(* CoDeSys 2.3 project: cy-02-wg-030.pro *)
(* Title: cy-02-wg - Albino Infanzia E10 *)
(* Author: Andrea Ravasio *)
(* Libraries: Standard.lib 2.12.10 14:48:34, Util.lib 26.9.14 10:12:46, Visual.lib 2.12.10 14:48:34, WagoLibIdent.lib 25.2.13 11:12:16, WagoLibStatus.lib 2.12.10 14:48:32, SysLibFile.lib 2.12.10 14:48:34, SysLibRtc.lib 2.12.10 14:48:32, SysLibSockets.lib 10.2.11 09:20:54, SysLibEvent.lib 2.12.10 14:48:34, SysLibPlcCtrl.lib 2.12.10 14:48:32, SysLibCallback.lib 2.12.10 14:48:32, serial_interface_01.lib 22.4.13 12:50:14, SerComm.lib 31.5.11 08:54:36, MBus_03.lib 9.2.13 17:51:58, mod_com.lib 2.12.10 14:48:32, Modb_l05.lib 22.4.13 12:50:12 *)

(* PLC configuration (modules and I/O channels)
0750-1506 8DI / 8DO 24V DC 0.5A [Type_34_8_Channels] node 0, in %IB12 out %QB8 {INTTypePAAssignment = PLC; INTTypeModule = plugged}
  CIR06_AL AT %IX6.0 [BOOLOnX_I] Ch_1 Digital input
  CIR06_EN AT %QX4.0 [BOOLOnX_Q] 9 - Ch_1 Digital output
  CIR06_ST AT %IX6.1 [BOOLOnX_I] Ch_2 Digital input
  CIR06_ECO AT %QX4.1 [BOOLOnX_Q] 10 - Ch_2 Digital output
  CIR05_AL AT %IX6.2 [BOOLOnX_I] Ch_3 Digital input
  CIR05_EN AT %QX4.2 [BOOLOnX_Q] 11 - Ch_3 Digital output
  CIR06_AUTO AT %IX6.3 [BOOLOnX_I] Ch_4 Digital input
  CIR05_ECO AT %QX4.3 [BOOLOnX_Q] 12 - Ch_4 Digital output
  CIR04_AL AT %IX6.4 [BOOLOnX_I] Ch_5 Digital input
  CIR04_EN AT %QX4.4 [BOOLOnX_Q] 13 - Ch_5 Digital output
  CIR05_ST AT %IX6.5 [BOOLOnX_I] Ch_6 Digital input
  CIR04_ECO AT %QX4.5 [BOOLOnX_Q] 14 - Ch_6 Digital output
  CIR03_AL AT %IX6.6 [BOOLOnX_I] Ch_7 Digital input
  CIR03_EN AT %QX4.6 [BOOLOnX_Q] 15 - Ch_7 Digital output
  CIR05_AUTO AT %IX6.7 [BOOLOnX_I] Ch_8 Digital input
  CIR03_ECO AT %QX4.7 [BOOLOnX_Q] 16 - Ch_8 Digital output
0750-1506 8DI / 8DO 24V DC 0.5A [Type_34_8_Channels] node 1, in %IB12 out %QB8 {INTTypePAAssignment = PLC; INTTypeModule = plugged}
  CTL01_ST AT %IX6.8 [BOOLOnX_I] Ch_1 Digital input
  DOOR2_EN AT %QX4.8 [BOOLOnX_Q] 9 - Ch_1 Digital output
  DOOR2_ST AT %IX6.9 [BOOLOnX_I] Ch_2 Digital input
  CIR01_EN AT %QX4.9 [BOOLOnX_Q] 10 - Ch_2 Digital output
  CIR01_AL AT %IX6.10 [BOOLOnX_I] Ch_3 Digital input
  CIR02_EN AT %QX4.10 [BOOLOnX_Q] 11 - Ch_3 Digital output
  CIR01_ST AT %IX6.11 [BOOLOnX_I] Ch_4 Digital input
  AT %QX4.11 [BOOLOnX_Q] 12 - Ch_4 Digital output
  CIR03_ST AT %IX6.12 [BOOLOnX_I] Ch_5 Digital input
  AT %QX4.12 [BOOLOnX_Q] 13 - Ch_5 Digital output
  CIR01_AUTO AT %IX6.13 [BOOLOnX_I] Ch_6 Digital input
  AT %QX4.13 [BOOLOnX_Q] 14 - Ch_6 Digital output
  CIR02_AL AT %IX6.14 [BOOLOnX_I] Ch_7 Digital input
  AT %QX4.14 [BOOLOnX_Q] 15 - Ch_7 Digital output
  CIR02_ST AT %IX6.15 [BOOLOnX_I] Ch_8 Digital input
  AT %QX4.15 [BOOLOnX_Q] 16 - Ch_8 Digital output
0750-1506 8DI / 8DO 24V DC 0.5A [Type_34_8_Channels] node 2, in %IB13 out %QB9 {INTTypePAAssignment = PLC; INTTypeModule = plugged}
  KEY_CT_ST AT %IX7.0 [BOOLOnX_I] Ch_1 Digital input
  KEY_CT_EN AT %QX5.0 [BOOLOnX_Q] 9 - Ch_1 Digital output
  GZB_ST AT %IX7.1 [BOOLOnX_I] Ch_2 Digital input
  GZB_CTRL AT %QX5.1 [BOOLOnX_Q] 10 - Ch_2 Digital output
  VPN_OUT2 AT %IX7.2 [BOOLOnX_I] Ch_3 Digital input
  VPN_DIS AT %QX5.2 [BOOLOnX_Q] 11 - Ch_3 Digital output
  CIR04_AUTO AT %IX7.3 [BOOLOnX_I] Ch_4 Digital input
  AT %QX5.3 [BOOLOnX_Q] 12 - Ch_4 Digital output
  KEY_QE_ST AT %IX7.4 [BOOLOnX_I] Ch_5 Digital input
  AT %QX5.4 [BOOLOnX_Q] 13 - Ch_5 Digital output
  CIR03_AUTO AT %IX7.5 [BOOLOnX_I] Ch_6 Digital input
  AT %QX5.5 [BOOLOnX_Q] 14 - Ch_6 Digital output
  CIR02_AUTO AT %IX7.6 [BOOLOnX_I] Ch_7 Digital input
  TEST1 AT %QX5.6 [BOOLOnX_Q] 15 - Ch_7 Digital output
  CIR04_ST AT %IX7.7 [BOOLOnX_I] Ch_8 Digital input
  TEST2 AT %QX5.7 [BOOLOnX_Q] 16 - Ch_8 Digital output
0750-0650/0003-0000#03 RS 232 C Interface (Adjustable), 3 Byte [Type_21_1_Channels] node 3, in %IB8 out %QB8 {INTTypePAAssignment = PLC; INTTypeModule = plugged}
  AT %IX0.0 [BOOLOnX_I] Transmission acknowledgement
  AT %IX0.1 [BOOLOnX_I] Reception request
  AT %IX0.2 [BOOLOnX_I] Initialization acknowledgement
  AT %IX0.3 [BOOLOnX_I] Input buffer is full
  AT %IX0.4 [BOOLOnX_I] Number of received characters Bit 0
  AT %IX0.5 [BOOLOnX_I] Number of received characters Bit 1
  AT %IX0.6 [BOOLOnX_I] Number of received characters Bit 2
  AT %IB1 [BYTEOnB_I] Input data Byte 0
  AT %IB2 [BYTEOnB_I] Input data Byte 1
  AT %IB3 [BYTEOnB_I] Input data Byte 2
  AT %QX0.0 [BOOLOnX_Q] Transmission request
  AT %QX0.1 [BOOLOnX_Q] Reception acknowledgement
  AT %QX0.2 [BOOLOnX_Q] Initialization request
  AT %QX0.4 [BOOLOnX_Q] Number of characters Bit 0
  AT %QX0.5 [BOOLOnX_Q] Number of characters Bit 1
  AT %QX0.6 [BOOLOnX_Q] Number of characters Bit 2
  AT %QB1 [BYTEOnB_Q] Output data Byte 0
  AT %QB2 [BYTEOnB_Q] Output data Byte 1
  AT %QB3 [BYTEOnB_Q] Output data Byte 2
0750-0650/0003-0000#03 RS 232 C Interface (Adjustable), 3 Byte [Type_21_1_Channels] node 4, in %IB8 out %QB8 {INTTypePAAssignment = PLC; INTTypeModule = plugged}
  AT %IX2.0 [BOOLOnX_I] Transmission acknowledgement
  AT %IX2.1 [BOOLOnX_I] Reception request
  AT %IX2.2 [BOOLOnX_I] Initialization acknowledgement
  AT %IX2.3 [BOOLOnX_I] Input buffer is full
  AT %IX2.4 [BOOLOnX_I] Number of received characters Bit 0
  AT %IX2.5 [BOOLOnX_I] Number of received characters Bit 1
  AT %IX2.6 [BOOLOnX_I] Number of received characters Bit 2
  AT %IB5 [BYTEOnB_I] Input data Byte 0
  AT %IB6 [BYTEOnB_I] Input data Byte 1
  AT %IB7 [BYTEOnB_I] Input data Byte 2
  AT %QX2.0 [BOOLOnX_Q] Transmission request
  AT %QX2.1 [BOOLOnX_Q] Reception acknowledgement
  AT %QX2.2 [BOOLOnX_Q] Initialization request
  AT %QX2.4 [BOOLOnX_Q] Number of characters Bit 0
  AT %QX2.5 [BOOLOnX_Q] Number of characters Bit 1
  AT %QX2.6 [BOOLOnX_Q] Number of characters Bit 2
  AT %QB5 [BYTEOnB_Q] Output data Byte 0
  AT %QB6 [BYTEOnB_Q] Output data Byte 1
  AT %QB7 [BYTEOnB_Q] Output data Byte 2
0750-0461 2 AI PT100 (RTD) [Type_44_2_Channels] node 5, in %IB12 out %QB12 {INTTypePAAssignment = PLC; INTTypeModule = plugged}
  T_S02 AT %IW4 [INTOnW_I] Ch_1 signed Input value
  T_S01 AT %IW5 [INTOnW_I] Ch_2 signed Input value
Fieldbus variables [FB_VARS] node 1, in %IB0 out %QB0
Flag variables [FLAG_VARS] node 2, in %IB0 out %QB0
Modbus-Master [MB_MASTER] node 3, in %IB0 out %QB0
*)

(* Global variable list: Global_Constants *)
VAR_GLOBAL CONSTANT

	Plant_NAME			: STRING :='cySN:2 cyVER:30 - Albino Infanzia E10';
	Plant_SN			: DWORD  :=2;  		(* S/N Impianto di telecontrollo *)
	Plant_SW_VER		: WORD   :=30;		(* Versione SW installata *)

	(* Parameters *)
	Plant_DefaultTAmb	: INT	:=100;		(* [.1°C] Temperatura ambiente di default in caso di rottura sonda *)
	Plant_MaxRunTAmb	: INT   :=250; 		(* [.1°C] Temperatura ambiente massima funzionamento impianto *)
	Plant_AntiFreezeTAmb: INT   :=-40;		(* [.1°C] Antifreeze temperature, start circulators *)
	Plant_VRD_TAlarm	: INT   :=450; 		(* [.1°C] Temperatura di allarme VRD, blocco *)
	Plant_VRD_TMax		: INT   :=430; 		(* [.1°C] Setpoint massimo per uscita VRD *)
	Plant_VRD_TDefault	: INT	:=300;		(* [.1°C] Temperatura di default in caso di errore climatica *)
	Plant_CirOffDelay	: TIME	:=T#15m;	(* (Def.T#15m) Ritardo spegnimento pompe per ricircolo caldaia *)
	Plant_MaxWaterLoss	: WORD  :=2;		(* [lt/h] Massima perdita del circuito *)

	(* Filesystem *)
	FilesPath  			: STRING :='S:\';

	(* TCP Logger *)
	Logger_SERVER		: STRING:='';
	Logger_IP			: STRING:='192.168.100.3';
	Logger_PORT			: WORD  :=80;
	Logger_GETSTART		: STRING:='GET /cygmsrv/hsgm.ashx?';
	Logger_GETEND		: STRING:='$R$N$R$N';
	Logger_CHECK		: STRING:='True';
	Logger_CRLF			: STRING:='$R$N';
	Logger_DataFile		: STRING:='S:\LOG.DAT';
	Logger_DataFileOld	: STRING:='S:\LOG.BCK';
	Logger_IndexFile	: STRING:='S:\LOG.IDX';
	Logger_ConnRetries	: BYTE:=5;
	Logger_RecoverMsgs	: BYTE:=100;

	(* TCP Remote *)
	Remote_PORT			: WORD  :=10;
	Remote_WELCOME		: STRING:='Connected$R$N';
	Remote_OK			: STRING:='OK$R$N';
	Remote_ERROR		: STRING:='ERROR$R$N';

	(* TCP Sockets *)
	MAX_SEND_TCP_SERVER					 : DWORD:=3000;(*60000*)
	MAX_RECEIVE_TCP_SERVER				 : DWORD:=3000;
	MAX_RECEIVE_TCP_SERVER_SOCKET	 	 : DWORD:=1500;
	MAX_SEND_TCP_CLIENT					 : DWORD:=3000;(*15000*)
	MAX_RECEIVE_TCP_CLIENT				 : DWORD:=1500;
	MAX_RECEIVE_TCP_CLIENT_SOCKET		 : DWORD:=1500;
	MAX_RECEIVE_UDP_SERVER				 : INT  :=1472;
	MAX_RECEIVE_UDP_CLIENT				 : INT  :=1472;
	CONNECT_WATCHDOG_TIME				 : TIME :=t#10s;

	(* VISU COLORS *)
	COLOR_RED 		: DWORD:=16#2020F0;
	COLOR_YELLOW	: DWORD:=16#20F0F0;
	COLOR_GREEN		: DWORD:=16#20F020;
	COLOR_GREEN_OFF : DWORD:=16#006000;
	COLOR_LBLUE		: DWORD:=16#F0F080;

END_VAR

(* Global variable list: Global_Retain *)
VAR_GLOBAL RETAIN PERSISTENT
	GRU01_Clima : typ_Clima;
	CTL01_Count : DWORD;

	Mode_Manual : BOOL := FALSE;
END_VAR

(* Global variable list: Global_Variables *)
VAR_GLOBAL

	SYS    : typ_SYS;

	MODB01 : obj_MODBUS				:= ( ID:=1 , COM:=3, BAUDRATE:=BAUD_19200 );
	GRU01  : obj_MODBUS_ROBUR_DDC	:= ( ID:=1 , NetID:=479 );
	PDC01  : obj_PDC_ROBUR_GAHP		:= ( ID:=1 , NetID:=0 );
	CAL01  : obj_CAL_ROBUR_AY		:= ( ID:=1 , NetID:=1 );
	CAL02  : obj_CAL_ROBUR_AY		:= ( ID:=2 , NetID:=2 );

	TPV01  : obj_TPV				:= ( ID:=1 ); (* T_S01 - T_Amb *)
	TPV02  : obj_TPV				:= ( ID:=2 , IN_WMIN:=50 , IN_WMAX:=800 ); (* T_S02 *)
	TPV03  : obj_TPV				:= ( ID:=3 , IN_WMIN:=50 , IN_WMAX:=800 ); (* GRU01 - T_Send *)
	TPV04  : obj_TPV				:= ( ID:=4 , IN_WMIN:=50 , IN_WMAX:=800 ); (* GRU01 - T_Return *)
	TPV05  : obj_TPV				:= ( ID:=5 ); (* GRU01 - T_Amb *)
	T_AMB  : INT; (* From TPV01 *)

	CIR01  : obj_CIR				:= ( ID:=1 );
	CIR02  : obj_CIR				:= ( ID:=2 );
	CIR03  : obj_CIR				:= ( ID:=3 );
	CIR04  : obj_CIR				:= ( ID:=4 );
	CIR05  : obj_CIR				:= ( ID:=5 );
	CIR06  : obj_CIR				:= ( ID:=6 );

	CRON01 : obj_CRON				:= ( ID:=1 );
	CRON02 : obj_CRON				:= ( ID:=2 );
	CRON03 : obj_CRON				:= ( ID:=3 );
	CRON04 : obj_CRON				:= ( ID:=4 );
	CRON05 : obj_CRON				:= ( ID:=5 );
	CRON06 : obj_CRON				:= ( ID:=6 );
	CronEd : obj_CRON_EDITOR;

	CTL01  : obj_CTL				:= ( ID:=1 );

	MBUS01 : obj_MBUS				:= ( ID:=1 , COM:=2 , BAUDRATE:=BAUD_2400 );
	CTB01  : obj_MBUS_CTB			:= ( ID:=1 , ADDRESS:=0 );

	Logger : typ_Logger;

	(**** SIMULATION ONLY ****)
(*	CIR01_EN	:BOOL;
	CIR01_ST	:BOOL;
	CIR01_MAN	:BOOL;
	CIR01_AL	:BOOL:=TRUE;
	CIR03_EN	:BOOL;
	CIR03_ECO	:BOOL;
	CIR03_ST	:BOOL;
	CIR03_AL	:BOOL;
	CIR04_EN	:BOOL;
	CIR04_ECO	:BOOL;
	CIR04_ST	:BOOL;
	CIR04_AL	:BOOL;
	CIR05_EN	:BOOL;
	CIR05_ECO	:BOOL;
	CIR05_ST	:BOOL;
	CIR05_AL	:BOOL;
	CIR06_EN	:BOOL;
	CIR06_ECO	:BOOL;
	CIR06_ST	:BOOL;
	CIR06_AL	:BOOL;
	CTL01_ST	:BOOL;
	KEY_CT_ST	:BOOL;
	KEY_CT_EN	:BOOL;
	GZB_ST		:BOOL;
	GZB_CTRL	:BOOL;
	VPN_DIS		:BOOL;
	VPN_ST1		:BOOL:=TRUE;
	VPN_ST2		:BOOL;
	VPN_CTRL1	:BOOL;
	VPN_CTRL2	:BOOL;
	KEY_QE_ST	:BOOL:=TRUE;
(*	TEST1		:BOOL;	*)
	TEST2		:BOOL;
	T_S01		:INT:=100;
	T_S02		:INT:=100;
*)

END_VAR

(* Data type in Logger *)
TYPE en_Logger_ErrLev :
(
	EL_Log			:=0,
	EL_Wrn			:=1,
	EL_Alarm		:=2,
	EL_AlarmStop	:=3
);
END_TYPE

(* Data type in Logger *)
TYPE en_Logger_Status :
(
	S_Logger_UNKNOWN := 0,
	S_Logger_IDLE,
	S_Logger_WAITCONN,
	S_Logger_WAITTX,
	S_Logger_WAITRESP,
	S_Logger_ERROR
);
END_TYPE

(* Data type *)
TYPE en_SYS_Objects :
(
	EO_SYS		:=0,  (* PLC *)
	EO_VPN		:=1,  (* VPN *)
	EO_DOOR		:=2,  (* Door & access control *)

	EO_CAL		:=10, (* Caldaia *)
	EO_CIR		:=11, (* Circolatore *)
	EO_CRON		:=12, (* Crono-termostato *)
	EO_VRD		:=13, (* Valvola miscelatore pannelli *)
	EO_CTL		:=14, (* Contalitri *)
	EO_CTB		:=15, (* Contabilizzatore *)
	EO_TPV		:=16, (* Temperature probes values *)
	EO_PPV		:=17, (* Pressure probes values *)
	EO_PBV		:=18, (* Over-Pressure Alarms *)
	EO_TBV		:=19, (* Over-Temperature Alarms *)
	EO_PMV		:=20, (* Under-Pressure Alarms *)
	EO_GRU		:=21, (* Gruppo termico *)
	EO_PDC		:=22, (* Pompa di calore *)
	EO_SOL		:=23, (* Pannello solare termico *)
	EO_ESOL		:=24, (* Pannello solare fotovoltaico *)
	EO_GAS		:=25, (* Contatore GAS *)
	EO_PORT		:=26, (* Misuratore di portata *)
	EO_FPV		:=27, (* Flow probes values *)
	EO_ANZ		:=28, (* Analizzatore di rete *)
	EO_SCA		:=29, (* Signal Control Alarms *)
	EO_LUX		:=30, (* Base Illumination point *)
	EO_LUXM		:=31, (* Metered Illumination point *)
	EO_PSG		:=32, (* Sensore di passaggio *)
	EO_HVAC		:=33, (* Heating, Ventilating and Air Conditioning *)
	EO_HYGRV	:=34, (* Relative Humidity sensors value *)
	EO_COOV		:=35, (* Carbon Dioxide CO2 sensors value *)

	EO_ZGW			:=200,  (* ZigBee - Gateway *)
	EO_ZRM			:=201,	(* ZigBee - Repeater *)
	EO_ZREL			:=202,	(* ZigBee - Actuator rele *)
	EO_ZTHL			:=203,	(* ZigBee - Temperature Sensor *)

	EO_ASGW			:=250,	(* ASi - Gateway *)
	EO_ASCBI		:=251,	(* ASi - Input Board, Ciabatta *)

	EO_LON			:=1000, (* Bus - LON *)
	EO_MODBUS		:=1001, (* Bus - MODBUS *)
	EO_MBUS			:=1002, (* Bus - M-BUS *)
	EO_MODBUS_TCP	:=1003, (* Bus - MODBUS TCP *)

	EO_GENERIC		:=9000, (* Generic dataset *)
	EO_EXPO			:=9001  (* EXPO dataset *)
);
END_TYPE

(* Data type *)
TYPE en_SYS_Status :
(
	S_UNKNOWN  := 0,
	S_STARTUP,
	S_INIT_RTC,
	S_INIT_VAR,
	S_AUTOTEST,
	S_RUNNING,
	S_SHUTDOWN,
	S_HALT
);
END_TYPE

(* Data type in Plant_Objects *)
TYPE typ_Clima : (* CURVA CLIMATICA *)
STRUCT
	InitOK:		BOOL;
	Points: 	ARRAY [0..10] OF POINT;
END_STRUCT
END_TYPE

(* Data type in Plant_Objects *)
TYPE typ_Cron_Calendar :
STRUCT
	Profile		: ARRAY[0..384] OF BYTE;
END_STRUCT
END_TYPE

(* Data type in Plant_Objects *)
TYPE typ_Cron_Jolly :
STRUCT
	Start		: DT;
	End			: DT;
	Temp		: WORD;
	Flags		: WORD; (* B0:Enabled B1..B15:Unused *)
END_STRUCT
END_TYPE

(* Data type in Plant_Objects *)
TYPE typ_Cron_Profile :
STRUCT
	Flags		: WORD;
	Setpoint	: ARRAY [0..95] OF WORD;
END_STRUCT
END_TYPE

(* Data type in Logger *)
TYPE typ_Logger :
STRUCT
	Status		: en_Logger_Status;

	SendReq		: BOOL;
	SendIdx		: DWORD;
	SendData	: ARRAY [0..MAX_SEND_TCP_CLIENT] OF BYTE;
	SendLen		: DINT;

	TData		: ARRAY [0..MAX_SEND_TCP_CLIENT] OF BYTE;
	TLen		: DINT;

	LastIdxPos	: DWORD;

	(* Temporary variables used by objects *)
	s1			: STRING(256);
	i1			: WORD;

END_STRUCT
END_TYPE

(* Data type in Plant_Objects *)
TYPE typ_MODBUS_VAR : (* Gestione parametri MODBUS *)
STRUCT
	SlaveAddress	: BYTE;
	FunCode			: BYTE;
	FunAddress		: WORD;
	Refresh_Time	: BYTE; (* 0:No refresh x:Refresh in seconds *)
	Refresh_Cnt		: BYTE; (* INTERNAL *)
	Variable		: POINTER TO WORD;
	Variable_Size	: BYTE;
	Variable_Mirror : WORD; (* INTERNAL [Force refresh on read variables when <>0] *)
END_STRUCT
END_TYPE

(* Data type *)
TYPE typ_SYS :
STRUCT
	Status			: en_SYS_Status;
	Warning			: BOOL;
	Alarm			: BOOL;
	AlarmStop		: BOOL;

	Time_LogString	: STRING;
	Time_Year		: WORD;
	Time_Month		: BYTE;
	Time_Day		: BYTE;

	Time_CT_DT		: DT;
	Time_CT_Day		: WORD;
	Time_CT_Quarter	: BYTE;

	LastLogs_Idx	: BYTE;
	LastLogs_Dat	: ARRAY[0..5] OF STRING;
	LastLogs_Msg	: ARRAY[0..5] OF STRING;

END_STRUCT
END_TYPE

(* POU PLC_PRG, ST *)
PROGRAM PLC_PRG
VAR
	Timer1: TON; (* Fast controls tick *)
	Timer2: TON; (* Plant control tick *)
	Timer3: TON; (* Logger timer *)
END_VAR
(******************************************************************************
 ****                           MAIN TASK CODE                             ****
 ******************************************************************************

	Network setup:
		IP  = 192.168.100.2 | MSK = 255.255.255.0
		GW	= 192.168.100.1 | DNS = 192.168.100.1
		SNTP = 193.204.114.232 (3600s) ==> 192.168.100.3

*)

(*==============================*)
(*===== Main status machine ====*)
(*==============================*)
Main_Stm();

(*==============================*)
(*== Running cycle operations ==*)
(*==============================*)
IF SYS.Status>S_INIT_VAR THEN

	(* Execute MODBUS process *)
	MODB01();
	(* Execute M-BUS processes *)
	MBUS01();
	CTB01( MBus:=MBUS01.MBus );
	(*
	MBUS02();
	CTB02( MBus:=MBUS02.MBus );
	*)

END_IF

(*==============================*)
(*== System cycle operations ===*)
(*==============================*)
(* Execute TCP processes *)
Logger_Proc();
Remote_Proc();
(* Update user led *)
USRLED_Update();
(* Execute Cron Editor commands *)
CronEd();
(* External resources *)
   IF NOT TPV01.ERR THEN T_AMB:=T_S01;
ELSIF NOT TPV05.ERR THEN T_AMB:=GRU01.TAmb;
ELSE 					 T_AMB:=Plant_DefaultTAmb;
END_IF

(**** SIMULATION ONLY ****)
(*
CIR01_ST:=CIR01_EN XOR TEST2;
CIR03_ST:=CIR03_EN XOR TEST2;
CIR04_ST:=CIR04_EN XOR TEST2;
CIR05_ST:=CIR05_EN XOR TEST2;
CIR06_ST:=CIR06_EN XOR TEST2;
*)
END_PROGRAM
ACTION Main_Stm:
CASE Sys.Status OF

	S_STARTUP:
		Sys.Status:=S_INIT_RTC;

	S_INIT_RTC:
		(* Check RTC and update from network *)
		RTC_Update();
		(* Check time *)
		IF Sys.Time_Year>2000 THEN
			Sys.Status:=S_INIT_VAR;
		END_IF

	S_INIT_VAR:
		LogEv(EL_Wrn,EO_SYS,0,1,CONCAT('System_startup_v',WORD_TO_STRING(Plant_SW_VER)));
		Sys.Status:=S_RUNNING;

	S_RUNNING:
		Timer1(IN:=NOT Timer1.Q,PT:=T#50ms);
		IF Timer1.Q THEN
			(* Update meters *)
			CTL01 ( CTL_ST:=CTL01_ST, COUNT:=CTL01_Count );
			(* Update system checks *)
			SYS_Proc();
		END_IF

		Timer2(IN:=NOT Timer2.Q,PT:=T#500ms);
		IF Timer2.Q THEN
			(* Read current date/time *)
			RTC_Update();
			(* Execute plant operations *)
			TPV01	 ( IN:=T_S01 );
			TPV02	 ( IN:=T_S02 );
			TPV03	 ( IN:=GRU01.TSend );
			TPV04	 ( IN:=GRU01.TRet );
			TPV05	 ( IN:=GRU01.TAmb );
			(* CRON01   ( SETPOINT=>CIR01.Ctrl_SetPoint ); *) CRON01(); CIR01.CIR_RUN_REQ:=SEL(CRON01.SetPoint>180,FALSE,TRUE);
			(* CRON02   ( SETPOINT=>CIR02.Ctrl_SetPoint ); *) CRON02(); CIR02.CIR_RUN_REQ:=SEL(CRON02.SetPoint>180,FALSE,TRUE);
			CRON03   ( SETPOINT=>CIR03.Ctrl_SetPoint );
			CRON04   ( SETPOINT=>CIR04.Ctrl_SetPoint );
			CRON05   ( SETPOINT=>CIR05.Ctrl_SetPoint );
			CRON06   ( SETPOINT=>CIR06.Ctrl_SetPoint );
			CIR01    ( CIR_AL:=CIR01_AL , CIR_ST:=CIR01_ST , CIR_AUTO:=CIR01_AUTO , CIR_EN=>CIR01_EN );
			CIR02    ( CIR_AL:=CIR02_AL , CIR_ST:=CIR02_ST , CIR_AUTO:=CIR02_AUTO , CIR_EN=>CIR02_EN );
			CIR03    ( CIR_AL:=CIR03_AL , CIR_ST:=CIR03_ST , CIR_AUTO:=CIR03_AUTO , CIR_EN=>CIR03_EN );
			CIR04    ( CIR_AL:=CIR04_AL , CIR_ST:=CIR04_ST , CIR_AUTO:=CIR04_AUTO , CIR_EN=>CIR04_EN );
			CIR05    ( CIR_AL:=CIR05_AL , CIR_ST:=CIR05_ST , CIR_AUTO:=CIR05_AUTO , CIR_EN=>CIR05_EN );
			CIR06    ( CIR_AL:=CIR06_AL , CIR_ST:=CIR06_ST , CIR_AUTO:=CIR06_AUTO , CIR_EN=>CIR06_EN );
			GRU01.Run:=( CIR01.Run OR CIR03.Run OR CIR04.Run OR CIR05.Run OR CIR06.Run ) AND SYS.AlarmStop=FALSE;
			GRU01	 ( Clima:=GRU01_Clima, MODBUS:=MODB01 );
			PDC01	 ();
			CAL01	 ();
			CAL02	 ();
			(* Test toggle *)
			IF TEST1 THEN TEST1:=FALSE; ELSE TEST1:=TRUE; END_IF
		END_IF

		Timer3(IN:=NOT Timer3.Q,PT:=T#5m);
		IF Timer3.Q THEN
			(* Trig logger *)
			LogTrig();
			(* Execute temporary CSV logger *)
			CSV_Log();
		END_IF

	S_SHUTDOWN:
		(* Stop caldaia *)
		(* Stop deviatori *)
		(* Aspetta 5 min prima di spegnere eventuali circolatori *)
		Sys.Status:=S_STARTUP;

	S_HALT:
		(* Aspetta uscita manuale *)
		Sys.Status:=S_STARTUP;

ELSE
	Sys.Status:=S_STARTUP;
END_CASE;
END_ACTION

(* POU TCP_Logger/Logger_Proc, ST *)
PROGRAM Logger_Proc
VAR
	c1:         	TCPCLIENT;

	Open:	    	BOOL;
	IpAddr:			DWORD;
	InetAddr:		DWORD;
	Connected:  	BOOL;
	Error:      	DINT;
	TxTrig:     	BOOL;
	RxData:			ARRAY [0..MAX_RECEIVE_TCP_CLIENT] OF BYTE;
	RxLen:			DINT;

	Retry:			BYTE;	(* Counter for connection retries *)
	Recovered:		BYTE;	(* Counter for recovered unsent messages *)

	i:				DINT;
	pos:			DWORD;
	hFile:			DWORD;

END_VAR
(*=== State machine ===*)
CASE Logger.Status OF

	S_Logger_UNKNOWN:
		(* Startup *)
		Logger.SendReq:=FALSE;
		Open:=FALSE;
		Logger.Status:=S_Logger_IDLE;

	S_Logger_IDLE:
		(* Wait request *)
		IF Logger.SendReq THEN
			(* Resolve server name or use static IP *)
			IF LEN(Logger_SERVER)=0 THEN
				InetAddr:=SysSockInetAddr(Logger_IP);
			ELSE
				IpAddr:=SysSockGetHostByName(ADR(Logger_SERVER));
				DWORDSWAP(pIn:=ADR(IpAddr), pOut:=ADR(InetAddr));
			END_IF
			TxTrig:=FALSE;
			RxLen:=0;
			(* Open connection *)
			Open:=TRUE;
			Logger.Status:=S_Logger_WAITCONN;
		END_IF

	S_Logger_WAITCONN:
		(* Wait connection *)
		IF Connected THEN
			(* Send data *)
			TxTrig:=TRUE;
			Logger.Status:=S_Logger_WAITTX;
		END_IF
		IF Error>0 THEN
			Open:=FALSE;
			Logger.Status:=S_Logger_ERROR;
		END_IF

	S_Logger_WAITTX:
		(* Wait transmission *)
		IF NOT TxTrig THEN
			Logger.Status:=S_Logger_WAITRESP;
		END_IF
		IF Error>0 THEN
			Open:=FALSE;
			Logger.Status:=S_Logger_ERROR;
		END_IF

	S_Logger_WAITRESP:
		(* Wait response *)
		IF Connected=FALSE (* OR TIMEOUT!! *) THEN
			Open:=FALSE;
			(* Check response *)
			IF RxLen>=4 AND CHKSTRING(pString:=ADR(RxData), pPattern:=ADR(Logger_CHECK)) THEN
				Logger.SendReq:=FALSE;
				Retry:=0;
				(* Check unsent messages to flush *)
				IF Recovered<Logger_RecoverMsgs THEN
					MsgChk();
					IF Logger.SendReq=TRUE THEN
						Recovered:=Recovered+1;
					ELSE
						Recovered:=0;
					END_IF
				ELSE
					Recovered:=0;
				END_IF
				Logger.Status:=S_Logger_IDLE;
			ELSE
				Logger.Status:=S_Logger_ERROR;
			END_IF
		END_IF

	S_Logger_ERROR:
		(* Connection error or send failure *)
		Retry:=Retry+1;
		IF Retry>Logger_ConnRetries THEN
			(* Save message as unsent *)
			MsgSave();
			Logger.SendReq:=FALSE;
			Retry:=0;
		END_IF
		Logger.Status:=S_Logger_IDLE;

ELSE
	Logger.Status:=S_Logger_UNKNOWN;
END_CASE


(*=== Execute client lib ===*)
c1(
	xOpenConnection			:= Open,
	dwInetAddr 				:= InetAddr,
	wPortNumber				:= Logger_PORT,
	ptSendData				:= ADR(Logger.SendData),
	diSendCount				:= Logger.SendLen,
	tConnectWatchdogTime	:= t#10s,
	xStartSend				:= TxTrig,
	aReceiveBuffer			:= RxData,
	diReceiveCount			:= RxLen,
	xConnected				=> Connected,
	diError					=> Error
);

(*=== Process Rx data ===*)
(*IF RxLen>0 THEN
	RxLen:=0;
END_IF*)
END_PROGRAM
ACTION MsgChk:
(* Open index file *)
hFile:=SysFileOpen(Logger_IndexFile,'r');
IF hFile=0 THEN
	RETURN;
END_IF
(* Search oldest message to recover *)
SysFileSetPos(hFile,Logger.LastIdxPos);
Logger.SendLen:=0;
REPEAT
	SysFileRead(hFile, ADR(Logger.SendIdx), SIZEOF(Logger.SendIdx));
	pos:=SysFileGetPos(hFile);
	SysFileRead(hFile, ADR(Logger.SendLen), SIZEOF(Logger.SendLen));
UNTIL
	SysFileEOF(hFile) OR Logger.SendLen<>0
END_REPEAT
SysFileClose(hFile);
(* Delete index file when all messages are recovered *)
IF Logger.SendLen=0 THEN
	Logger.LastIdxPos:=0;
	SysFileDelete(Logger_IndexFile);
	RETURN;
END_IF
(* Recover message data *)
hFile:=SysFileOpen(Logger_DataFile,'r');
IF hFile<>0 THEN
	SysFileSetPos(hFile,Logger.SendIdx);
	SysFileRead(hFile,ADR(Logger.SendData),Logger.SendLen);
	Logger.SendReq:=TRUE;
	SysFileClose(hFile);
END_IF
(* Clear index entry *)
hFile:=SysFileOpen(Logger_IndexFile,'a');
IF hFile<>0 THEN
	SysFileSetPos(hFile,pos);
	i:=0;
	SysFileWrite(hFile, ADR(i), 4);
	Logger.LastIdxPos:=SysFileGetPos(hFile);
	SysFileClose(hFile);
END_IF
END_ACTION
ACTION MsgSave:
(* Add log position in recovery indexes *)
hFile:=SysFileOpen(Logger_IndexFile,'a');
SysFileWrite(hFile, ADR(Logger.SendIdx), SIZEOF(Logger.SendIdx));
SysFileWrite(hFile, ADR(Logger.SendLen), SIZEOF(Logger.SendLen));
SysFileClose(hFile);
END_ACTION

(* POU Utils Functions/TCPCLIENT, ST *)
FUNCTION_BLOCK TCPCLIENT
(***********************************************************************************************************	*)
(* Version: 1.3b                        			          													*)
(* Date: 28.10.2014                   				          							            			*)
(***********************************************************************************************************	*)
(* WAGO Kontakttechnik GmbH Hansastr. 27 32423 Minden(Westf.)													*)
(* Tel. +0049 571/887-0 Fax. +0049 571/887-0																	*)
(* Author: VB																									*)
(***********************************************************************************************************	*)
(*Description:	A TCP client to read and write data with additional connection watchdog							*)
(*History:																										*)
(*Version 1.3b: 28.10.2014: Use DWORD address for IP (Andrea Ravasio)											*)
(*Version 1.3: 11.02.2011: Changes according to 750-880/881											 			*)
(*Version 1.2: 29.08.2007 Bugfix TCP Client																		*)
(*Version 1.1: 15.01.2007 Changes according to FW11																*)
(*Version 1.0: 09.03.2006 Release																				*)
(***********************************************************************************************************	*)
VAR CONSTANT
	STATE_CREATE     				 : BYTE:= 0;
	STATE_OPEN     					 : BYTE:= 1;
	STATE_IOCTL    					 : BYTE:= 2;
	STATE_CONNECT     				 : BYTE:= 10;
	STATE_TX       					 : BYTE:= 20;
	STATE_RX       					 : BYTE:= 30;
	STATE_CLOSE    					 : BYTE:= 40;
	STATE_ERROR_TRAP			     : BYTE:= 200;
END_VAR

VAR_INPUT
	xOpenConnection					: BOOL;
	dwInetAddr						: DWORD; (* <== Use SysSockInetAddr() value or
													swapped bytes order of SysSockGetHostByName() value *)
	wPortNumber						: WORD;
	ptSendData						: POINTER TO ARRAY[0..MAX_SEND_TCP_CLIENT] OF BYTE;
	diSendCount						: DINT;
	tConnectWatchdogTime		    : TIME := t#10s;
END_VAR
VAR_OUTPUT
	xConnected						: BOOL;
	diError 						: DINT := 0;
END_VAR
(* ErrorCodes -----------------------------------------
	16#8001 => No socket descriptor available 
	16#8002 => SysSockSend returns -1 
	16#8003 => Socket was "gracefully closed" 
	16#8004 => switching to none blocking mode fails
	16#8005 => SysSockClose() returns FALSE 
    16#8006 => SysSockConnect() fails
    16#8007 => SysSockSend() fails
	16#8008 => error state machine 
	16#8009 => timeout while waiting for data from server 
------------------------------------------------------------*)
VAR_IN_OUT
	xStartSend							: BOOL;
	aReceiveBuffer						: ARRAY [0..MAX_RECEIVE_TCP_CLIENT] OF BYTE;
	diReceiveCount						: DINT;
END_VAR
VAR
	m_State								: BYTE := 0;
	m_ReceiveBuffer						: ARRAY [0..MAX_RECEIVE_TCP_CLIENT_SOCKET] OF BYTE;
	m_Socket							: DINT;
	m_AddressInfo						: SOCKADDRESS;
	m_BytesReceived						: DINT;
	m_diReturn							: DINT;
	m_xReturn							: BOOL;
	m_IoCtlParameter  					: DINT := 1; (* IOCTL-Parameter for non-blocking mode of sockets *)
	i									: INT;
	T_Connect							: TON;
	m_count								: DINT;
	diOption							: DINT := 1;
	m_Blocking   						: DINT := 0;
END_VAR
IF xOpenConnection THEN
	(* State maschine *)
	CASE  m_State OF

	(* -------------------------------------------------------------------------*)
	STATE_CREATE:
			(* create socket descriptor*)
			m_Socket := SysSockCreate(diAddressFamily	:= SOCKET_AF_INET,
													 diType		:= SOCKET_STREAM,
													 diProtocol := SOCKET_IPPROTO_TCP);
			IF m_Socket >= 0 THEN
			(*Set Push-Bit*)
				IF ADR(%MW0)=16#30000000  OR ADR(%MW0)=16#20000000 THEN (*841 or 881*)
					SysSockSetOption(
						diSocket:=m_Socket,
						diLevel:=6,
						diOption:=SOCKET_TCP_NODELAY,
						pOptionValue:=ADR(diOption),
						diOptionLength:=SIZEOF(diOption));
				ELSE
						;
				END_IF
				m_State := STATE_IOCTL; (* succesful *)
			ELSE
				diError := 16#8001;  (* no socket descriptor available *)
				m_State := STATE_ERROR_TRAP;
			END_IF

	(* -------------------------------------------------------------------------*)
	STATE_IOCTL: (* change  socket mode  to none blocking *)
		m_diReturn := SysSockIoctl( m_Socket, SOCKET_FIONBIO, ADR(m_IoCtlParameter));
		IF m_diReturn <> 0 THEN
			m_AddressInfo.sin_family := SOCKET_AF_INET;
			m_AddressInfo.sin_port := SysSockNtohs(wPortNumber);
			m_AddressInfo.sin_addr := dwInetAddr;
			m_State := STATE_CONNECT;
		ELSE
			diError := 16#8004;  (* switching to none blocking mode fails *)
			m_State := STATE_ERROR_TRAP;
		END_IF


	(* -------------------------------------------------------------------------*)
	STATE_CONNECT: (* connect with server *)
		T_Connect(IN:=TRUE , PT:=tConnectWatchdogTime);(*activate watchdog for establishing connection to a server*)
		m_xReturn := SysSockConnect ( m_Socket, ADR(m_AddressInfo),  SIZEOF(m_AddressInfo));
		IF m_xReturn THEN (* succesful *)
			IF xStartSend THEN
				m_State := STATE_TX;(*transmit data*)
			ELSE
				m_State := STATE_RX;(*wait for data from server*)
			END_IF
			xConnected:=TRUE;
			T_Connect(IN:=FALSE);
		ELSE
			IF T_Connect.Q THEN
				diError := 16#8006;  (* connect fails *)
				xConnected:=FALSE;
				T_Connect(IN:=FALSE);
				m_State := STATE_ERROR_TRAP;
				SysSockClose( m_Socket);
			ELSE
				m_State := STATE_CONNECT;(*client still  tries to set up connection*)
			END_IF
		END_IF


	STATE_TX:	 (* send TCP-message *)
		m_diReturn := SysSockSend(diSocket := m_Socket,
								  pbyBuffer := ADR(ptSendData^[0]),
								  diBufferSize := diSendCount-m_count,
								  diFlags := 0);

		CASE m_diReturn OF
		-1:	(* ERROR *)
			T_Connect(IN:=TRUE , PT:=CONNECT_WATCHDOG_TIME);(*activate watchdog to check communication*)
			IF t_Connect.Q THEN
				diError := 16#8007;
				T_Connect(IN:=FALSE);
				m_State:=STATE_CLOSE;
			END_IF
		0: (* socket was "gracefully closed" *)
			m_State := STATE_CLOSE;
			diError := 16#8003;
		ELSE (* succesful *)
			m_count:=m_count+m_diReturn;
			IF m_count>=diSendCount THEN
				diError := 16#0000;
				m_State := STATE_RX;
				m_count:=0;
				xStartSend:=FALSE;
			END_IF
			T_Connect(IN:=FALSE);
		END_CASE

	(* -------------------------------------------------------------------------*)
	STATE_RX: (* process receive data *)
			m_BytesReceived := SysSockRecv(	diSocket 	:= m_Socket,
										pbyBuffer 	:= ADR(m_ReceiveBuffer),		(* Address of receive buffer *)
										diBufferSize:= SIZEOF(m_ReceiveBuffer),
										diFlags		:= 0);

			CASE m_BytesReceived OF
			-1:	(* No data available or error occured *)
				T_Connect(IN:=TRUE , PT:=tConnectWatchdogTime);(*activate watchdog to check communication*)
				IF t_Connect.Q THEN
					diError:=16#8009;
					T_Connect(IN:=FALSE);
					m_State:=STATE_CLOSE;
				END_IF
				IF xStartSend THEN
					m_State:=STATE_TX	;(* WAIT IN THIS STATE  and check for arriving data or new send command*)
				END_IF;
			0: (* socket was "gracefully closed"  *)
				m_State:=STATE_CLOSE;
				diError := 16#8003;
			ELSE (* succesful *)
				diError := 16#0000;
				T_Connect(IN:=FALSE);
				(* Copy received data into receive buffer *)
				FOR i:= 0 TO DINT_TO_INT(m_BytesReceived	)-1 DO
					aReceiveBuffer[diReceiveCount]:= m_ReceiveBuffer[i];
					diReceiveCount:=(diReceiveCount+1) MOD SIZEOF(aReceiveBuffer);
				END_FOR

			END_CASE

	(* -------------------------------------------------------------------------*)
	STATE_CLOSE : (* close socket *)
		IF ADR(%MW0)=16#30000000  OR ADR(%MW0)=16#20000000 THEN (*841 or 881*)
			;
		ELSE
			SysSockShutdown(m_Socket, 0);;(*870*)
		END_IF
		m_xReturn := SysSockClose( m_Socket);
		m_Socket := -1;
		m_State := 0; (* succesful *)
		xConnected:=FALSE;
		T_Connect(IN:=FALSE);
	(* -------------------------------------------------------------------------*)
	STATE_ERROR_TRAP: (* error handling *)
		xConnected:=FALSE;

	ELSE  (* Bad FSM code trap  *)
			m_State:= STATE_ERROR_TRAP;
			diError:= 16#8008;
	END_CASE

ELSE(*close connection*)
	IF m_Socket >= 0 THEN
		IF ADR(%MW0)=16#30000000  OR ADR(%MW0)=16#20000000 THEN (*841 or 881*)
			;
		ELSE
			SysSockShutdown(m_Socket, 0);;(*870*)
		END_IF
		SysSockClose( m_Socket);
	END_IF
	m_Socket := -1;
	diError := 16#0000;
	m_State := STATE_CREATE;
	xConnected:=FALSE;
	T_Connect(IN:=FALSE);
END_IF
END_FUNCTION_BLOCK

(* POU Utils Functions/DWORDSWAP, ST *)
FUNCTION DWORDSWAP:BOOL
VAR_INPUT
	pIn:POINTER TO ARRAY[1..4] OF BYTE;
	pOut:POINTER TO ARRAY[1..4] OF BYTE;
END_VAR
VAR
END_VAR
pOut^[1]:=pIn^[4];
pOut^[2]:=pIn^[3];
pOut^[3]:=pIn^[2];
pOut^[4]:=pIn^[1];
END_FUNCTION

(* POU Utils Functions/CHKSTRING, ST *)
FUNCTION CHKSTRING : BOOL
VAR_INPUT
	pString: POINTER TO BYTE;
	pPattern: POINTER TO BYTE;
END_VAR
VAR
END_VAR
CHKSTRING:=TRUE;
WHILE pPattern^<>0 AND CHKSTRING DO
	IF pPattern^<>pString^ THEN CHKSTRING:=FALSE; END_IF
	pString:=pString+1;
	pPattern:=pPattern+1;
END_WHILE
END_FUNCTION

(* POU TCP_Remote/Remote_Proc, ST *)
PROGRAM Remote_Proc
VAR
	s1:         	TCPSERVER;
	Enable: 		BOOL;
	Connected: 		BOOL;
	Error: 			DINT;

	TxData:			ARRAY [0..MAX_SEND_TCP_SERVER] OF BYTE;
	TxLen:			DINT;
	TxTrig:			BOOL;

	RxData:			ARRAY [0..MAX_RECEIVE_TCP_SERVER] OF BYTE;
	RxLen:			DINT;

	Status:			DINT;

	(* Command interpreter *)

	Cmd_Buf:		ARRAY [0..MAX_RECEIVE_TCP_SERVER] OF BYTE;
	Cmd_Buf_U16:	POINTER TO WORD;
	Cmd_Buf_INT:	POINTER TO INT;
	Cmd_BufLen:		WORD;
	Cmd_St:			WORD;

	Cmd_Obj:		WORD;
	Cmd_ObjIdx:		WORD;
	Cmd_C:			WORD;
	Cmd_R:			WORD;
	Cmd_CLen:		WORD;
	Cmd_RLen:		WORD;

	i : WORD;
	j : INT;
	(*s2 : STRING;*)

END_VAR
(*=== State machine ===*)
CASE Status OF
	0: (* Startup *)
		TxLen:=0; TxTrig:=FALSE;
		RxLen:=0;
		Enable:=TRUE;
		Status:=1;

	1: (* Wait incoming connection *)
		IF Connected THEN
			(* Log access *)(*
			LogEv(EL_Log,EO_VPN,1,5,'Remote');*)
			(* Send welcome message *)(*
			ADDSTRING(pTxData:=ADR(TxData), pString:=ADR(Remote_WELCOME), TxLen:=TxLen);
			TxTrig:=TRUE;*)
			(* Reset vars *)
			Cmd_BufLen:=0;
			Cmd_St:=0;
			Status:=2;
		END_IF
		IF Error>1 THEN
			Enable:=FALSE;
			Status:=0;
		END_IF

	2: (* Wait command *)
		IF RxLen>0 THEN
			(*=== Interpreter start ===*)
			IF Cmd_BufLen+(RxLen/2)>=MAX_RECEIVE_TCP_SERVER THEN
				(* ERROR *)
				Cmd_BufLen:=0;
			ELSE
				i:=HEXTORAW(pString:=ADR(RxData), StringLen:=DINT_TO_WORD(RxLen), pData:=ADR(Cmd_Buf[Cmd_BufLen]));
				Cmd_BufLen:=Cmd_BufLen+i;
			END_IF
			IF Cmd_BufLen>=8 THEN
				Cmd_Buf_U16:=ADR(Cmd_Buf[6]);
				IF Cmd_BufLen>=(8+Cmd_Buf_U16^) THEN
					Cmd_CLen:=Cmd_Buf_U16^;
					Cmd_Buf_U16:=ADR(Cmd_Buf[0]); Cmd_Obj:=Cmd_Buf_U16^;
					Cmd_Buf_U16:=ADR(Cmd_Buf[2]); Cmd_ObjIdx:=Cmd_Buf_U16^;
					Cmd_Buf_U16:=ADR(Cmd_Buf[4]); Cmd_C:=Cmd_Buf_U16^;
					(* Log command *)(*
					s2:='RCmd_';		s2:=CONCAT(s2,WORD_TO_STRING(Cmd_Obj));
					s2:=CONCAT(s2,'_'); s2:=CONCAT(s2,WORD_TO_STRING(Cmd_ObjIdx));
					s2:=CONCAT(s2,'_'); s2:=CONCAT(s2,WORD_TO_STRING(Cmd_C));
					s2:=CONCAT(s2,'_');	s2:=CONCAT(s2,WORD_TO_STRING(Cmd_CLen));
					LogEv(EL_Log,EO_VPN,1,6,s2);*)
					(* Execute command *)
					Command();
					Cmd_BufLen:=0;
				END_IF
			END_IF
			(*=== Interpreter end ===*)
			RxLen:=0;
		END_IF
		IF NOT Connected THEN
			Status:=0;
		END_IF

ELSE
	Status:=0;
END_CASE


(*=== Execute server lib ===*)
s1(
	xEnable				:= Enable,
	wPortNumber			:= Remote_PORT,
	tServerTimeOut		:= t#15m,
	ptSendData			:= ADR(TxData),
	diSendCount			:= TxLen,
	xStartSend			:= TxTrig,
	aReceiveBuffer		:= RxData,
	diReceiveCount		:= RxLen,
	xClientConnected	=> Connected,
	diError				=> Error
);
END_PROGRAM
ACTION Cmd_CAL:
(* Check index *)
IF Cmd_ObjIdx<1 OR Cmd_ObjIdx>2 THEN
	Cmd_R:=2;
	RETURN;
END_IF

(* Process command *)
CASE Cmd_C OF

	3: (* TRY REARM *)
		IF Cmd_ObjIdx=1 THEN
			CAL01.Rearm:=TRUE;
		ELSE
			CAL02.Rearm:=TRUE;
		END_IF

ELSE
	Cmd_R:=3;
END_CASE
END_ACTION
ACTION Cmd_CRON:
(* Check index *)
IF Cmd_ObjIdx<1 OR Cmd_ObjIdx>6 THEN
	Cmd_R:=2;
	RETURN;
END_IF

(* Process command *)
CASE Cmd_C OF

	1: (* GET PROFILE *)
		IF Cmd_CLen<>3 THEN
			Cmd_R:=4;
		ELSE
			(* Load profile *)
			CronEd.CN_Sel:=WORD_TO_BYTE(Cmd_ObjIdx);
			Cmd_Buf_U16:=ADR(Cmd_Buf[8]);
			CronEd.CN_YSel:=Cmd_Buf_U16^;
			CronEd.PR_Sel:=Cmd_Buf[10];
			CronEd.PR_Load_Exe();
			(* Copy data *)
			Cmd_RLen:=192;
			TxLen:=TxLen+RAWTOHEX(ADR(CronEd.PR.Setpoint),192,ADR(TxData[TxLen]));
		END_IF

	2: (* SET PROFILE *)
		IF Cmd_CLen<>(3+192) THEN
			Cmd_R:=4;
		ELSE
			(* Save profile *)
			CronEd.CN_Sel:=WORD_TO_BYTE(Cmd_ObjIdx);
			Cmd_Buf_U16:=ADR(Cmd_Buf[8]);
			CronEd.CN_YSel:=Cmd_Buf_U16^;
			CronEd.PR_Sel:=Cmd_Buf[10];
			MEMCPY(ADR(Cmd_Buf[11]),ADR(CronEd.PR.Setpoint),192);
			CronEd.PR_Save_Exe();
		END_IF

	5: (* GET CALENDAR MONTH *)
		IF Cmd_CLen<>3 THEN
			Cmd_R:=4;
		ELSE
			(* Load calendar *)
			CronEd.CN_Sel:=WORD_TO_BYTE(Cmd_ObjIdx);
			Cmd_Buf_U16:=ADR(Cmd_Buf[8]);
			CronEd.CN_YSel:=Cmd_Buf_U16^;
			CronEd.CA_Sel:=Cmd_Buf[10];
			CronEd.CA_Load_Exe();
			(* Copy data *)
			Cmd_RLen:=32;
			TxLen:=TxLen+RAWTOHEX(ADR(CronEd.CA.Profile),32,ADR(TxData[TxLen]));
		END_IF

	6: (* SET CALENDAR MONTH *)
		IF Cmd_CLen<>(3+32) THEN
			Cmd_R:=4;
		ELSE
			(* Save calendar *)
			CronEd.CN_Sel:=WORD_TO_BYTE(Cmd_ObjIdx);
			Cmd_Buf_U16:=ADR(Cmd_Buf[8]);
			CronEd.CN_YSel:=Cmd_Buf_U16^;
			CronEd.CA_Sel:=Cmd_Buf[10];
			MEMCPY(ADR(Cmd_Buf[11]),ADR(CronEd.CA.Profile),32);
			CronEd.CA_Save_Exe();
		END_IF

	9: (* CRON RESTART *)
		CASE Cmd_ObjIdx OF
			1: CRON01.InitOK:=FALSE;
			2: CRON02.InitOK:=FALSE;
			3: CRON03.InitOK:=FALSE;
			4: CRON04.InitOK:=FALSE;
			5: CRON05.InitOK:=FALSE;
			6: CRON06.InitOK:=FALSE;
		END_CASE

ELSE
	Cmd_R:=3;
END_CASE
END_ACTION
ACTION Cmd_GRU:
(* Check index *)
IF Cmd_ObjIdx<>1 THEN
	Cmd_R:=2;
	RETURN;
END_IF

(* Process command *)
CASE Cmd_C OF

	1: (* GET CLIMATIC *)
		Cmd_RLen:=20;
		FOR i:=0 TO 4 DO
			j:=DINT_TO_INT(GRU01_Clima.Points[i].X);
			TxLen:=TxLen+RAWTOHEX(ADR(j),2,ADR(TxData[TxLen]));
			j:=DINT_TO_INT(GRU01_Clima.Points[i].Y);
			TxLen:=TxLen+RAWTOHEX(ADR(j),2,ADR(TxData[TxLen]));
		END_FOR

	2: (* SET CLIMATIC *)
		IF Cmd_CLen<>20 THEN
			Cmd_R:=4;
		ELSE
			FOR i:=0 TO 4 DO
				Cmd_Buf_INT:=ADR(Cmd_Buf[8+4*i]); j:=Cmd_Buf_INT^;
				GRU01_Clima.Points[i].X:=INT_TO_DINT(j);
				Cmd_Buf_INT:=ADR(Cmd_Buf[10+4*i]); j:=Cmd_Buf_INT^;
				GRU01_Clima.Points[i].Y:=INT_TO_DINT(j);
			END_FOR
		END_IF

ELSE
	Cmd_R:=3;
END_CASE
END_ACTION
ACTION Cmd_PDC:
(* Check index *)
IF Cmd_ObjIdx<>1 THEN
	Cmd_R:=2;
	RETURN;
END_IF

(* Process command *)
CASE Cmd_C OF

	3: (* TRY REARM *)
		PDC01.Rearm:=TRUE;

ELSE
	Cmd_R:=3;
END_CASE
END_ACTION
ACTION Cmd_SYS:
(* Check index *)
IF Cmd_ObjIdx<>0 THEN
	Cmd_R:=2;
	RETURN;
END_IF

(* Process command *)
CASE Cmd_C OF

	0: (* ECHO *)
		IF Cmd_CLen<>0 THEN
			TxLen:=0;
		END_IF

	1: (* LOG REQUEST *)
		LogTrig();

	2: (* REARM *)
		Sys.Warning:=FALSE;
		Sys.Alarm:=FALSE;
		Sys.AlarmStop:=FALSE;

	3: (* GET INFO1 *)
		Cmd_RLen:=6;
		TxLen:=TxLen+RAWTOHEX(ADR(Plant_SN),4,ADR(TxData[TxLen]));
		TxLen:=TxLen+RAWTOHEX(ADR(Plant_SW_VER),2,ADR(TxData[TxLen]));

ELSE
	Cmd_R:=3;
END_CASE
END_ACTION
ACTION Command:
(* Default response OK/NODATA *)
Cmd_R:=0;
Cmd_RLen:=0;
TxLen:=16;

(* Check object *)
CASE Cmd_Obj OF

	EO_SYS:
		Cmd_SYS();

	EO_GRU:
		Cmd_GRU();

	EO_PDC:
		Cmd_PDC();

	EO_CAL:
		Cmd_CAL();

	EO_CRON:
		Cmd_CRON();

ELSE
	Cmd_R:=1;
END_CASE

(* Generate response *)
IF TxLen>0 THEN
	RAWTOHEX(ADR(Cmd_Obj)	,2,ADR(TxData[ 0]));
	RAWTOHEX(ADR(Cmd_ObjIdx),2,ADR(TxData[ 4]));
	RAWTOHEX(ADR(Cmd_R)		,2,ADR(TxData[ 8]));
	RAWTOHEX(ADR(Cmd_RLen)	,2,ADR(TxData[12]));
	TxTrig:=TRUE;
END_IF
END_ACTION

(* POU Utils Functions/TCPSERVER, ST *)
FUNCTION_BLOCK TCPSERVER
(***********************************************************************************************************	*)
(* Version: 1.6                                    			          											*)
(* Date: 11.02.2011                                   					          							    *)
(***********************************************************************************************************	*)
(* WAGO Kontakttechnik GmbH Hansastr. 27 32423 Minden(Westf.)													*)
(* Tel. +0049 571/887-0 Fax. +0049 571/887-0																	*)
(* Author: VB																									*)
(***********************************************************************************************************	*)
(*Description:	A TCP server to read and write data													       		*)
(*Historie:																										*)
(*Version 1.6: 11.02.2011: Changes according to 750-880/881											 			*)
(*Version 1.5: 27.11.2008 Bugfix allow reuse port																*)
(*Version 1.4: 13.10.2008 Bugfix transmitting large data														*)
(*Version 1.3: 15.01.2007 Changes according to FW11																*)
(*Version 1.2: 09.03.2006 Changes for socket handle 0											       			*)
(*Version 1.1: 14.02.2005 Release																				*)
(***********************************************************************************************************	*)
VAR CONSTANT
	STATE_INIT     				 : BYTE:= 0;
	STATE_OPEN     				 : BYTE:= 1;
	STATE_TX       				 : BYTE:= 20;
	STATE_RX       				 : BYTE:= 30;
	STATE_CLOSE    				 : BYTE:= 40;
	STATE_ERROR_TRAP		 	 : BYTE:= 200;
END_VAR
VAR_INPUT
	xEnable    					: BOOL;	 (* Set TRUE to enable function block *)
	wPortNumber					: WORD;  (* Port *)
	tServerTimeOut				: TIME:=t#50s;
	ptSendData					: POINTER TO ARRAY[0..MAX_SEND_TCP_SERVER] OF BYTE;
	diSendCount					: DINT;
END_VAR
VAR_OUTPUT
	xClientConnected  			: BOOL:= FALSE;
	diError 					: DINT:= 0;
END_VAR
(* Status Codes -----------------------------------------
	16#8001 => No socket descriptor available 
	16#8002 => SysSockBind fails 
	16#8003 => SysSockListen fails 
	16#8004 => switching to none blocking mode fails
	16#8005 => SysSockClose() returns FALSE 
    16#8006 => SysSockConnect() fails
    16#8007 => SysSockSend() fails
	16#8008 => error state machine 
	16#8009 => timeout while waiting for data from server 
	16#0001 => server waiting for client to establish connection
------------------------------------------------------------*)
VAR_IN_OUT
	xStartSend					: BOOL;
	aReceiveBuffer				: ARRAY [0..MAX_RECEIVE_TCP_SERVER] OF BYTE;
	diReceiveCount				: DINT;
END_VAR

VAR
	m_State    					: BYTE:= 0;
	m_ReceiveBuffer				: ARRAY [0..MAX_RECEIVE_TCP_SERVER_SOCKET] OF BYTE;
	m_ServerSocket				: DINT:= SOCKET_INVALID;
	m_Socket					: DINT:= SOCKET_INVALID;
	m_AddressInfo				: SOCKADDRESS;
	m_BytesReceived				: DINT;
	m_diReturn					: DINT;
	m_xReturn					: BOOL;
	m_SizeSockadr				: DWORD;
	m_ConnectionWatchdog		: TON;
	m_Flags						: DINT;
	m_NoneBlocking   			: DINT:= 1;
	m_Blocking   				: DINT:= 0;
	i							: INT;
	m_count						: DINT;
	diOption					: DINT := 1;
	on: DINT;
END_VAR
IF xEnable THEN
	CASE m_State OF
		STATE_INIT:
			(* Create Socket *)
			m_ServerSocket:= SysSockCreate( SOCKET_AF_INET, SOCKET_STREAM, 0);
			IF m_ServerSocket = SOCKET_INVALID THEN
				(* *)
				diError:= 16#8001;
				m_State:= STATE_ERROR_TRAP;
				RETURN;
			ELSE
				;
			END_IF
			(* Address bindings *)
			(********************)
			on:=1;
			SysSockSetOption( m_ServerSocket, SOCKET_SOL, SOCKET_SO_REUSEADDR, ADR(on), SIZEOF(on) );

			m_AddressInfo.sin_family:= SOCKET_AF_INET;
			m_AddressInfo.sin_port  := SysSockHtons( wPortNumber);
			m_AddressInfo.sin_addr  := SOCKET_INADDR_ANY;
			IF NOT SysSockBind( m_ServerSocket, ADR(m_AddressInfo), SIZEOF(m_AddressInfo)) THEN
				diError:= 16#8002;
				m_State:= STATE_ERROR_TRAP;
				RETURN;
			END_IF
			(* Wait for connections *)
			(************************)
			IF NOT SysSockListen( m_ServerSocket, 1) THEN
				diError:= 16#8003;
				m_State:= STATE_ERROR_TRAP;
			END_IF

			(* Puts SOCKET in NonBlocking mode *)
			m_diReturn:= SysSockIoctl( m_ServerSocket, SOCKET_FIONBIO, ADR(m_NoneBlocking));

			m_State:= STATE_OPEN;


		STATE_OPEN: 	(* Waiting for incomming connection *)
				m_SizeSockadr:=SIZEOF(m_AddressInfo);
				m_Socket:= SysSockAccept( m_ServerSocket, ADR(m_AddressInfo), ADR(m_SizeSockadr));
				diError:=State_open;
				IF m_Socket <> SOCKET_INVALID THEN
					xClientConnected:=TRUE;
					(*Set Push-Bit:new V1.5*)
					IF ADR(%MW0)=16#30000000  OR ADR(%MW0)=16#20000000 THEN (*841 or 881*)
						SysSockSetOption(
							diSocket:=m_Socket,
							diLevel:=6,
							diOption:=SOCKET_TCP_NODELAY,
							pOptionValue:=ADR(diOption),
							diOptionLength:=SIZEOF(diOption));
					ELSE
							;
					END_IF
					SysSockIoctl( m_Socket, SOCKET_FIONBIO, ADR(m_NoneBlocking));
					m_State:= STATE_RX;
					diError:=0;
				END_IF

		STATE_RX:
					m_BytesReceived:= SysSockRecv( m_Socket, ADR(m_ReceiveBuffer), SIZEOF(m_ReceiveBuffer), 0);
					CASE m_BytesReceived OF
					-1:(*no data available or error occured*)
						m_ConnectionWatchdog(IN:=TRUE , PT:=tServerTimeOut );
						IF m_connectionWatchdog.Q THEN
							m_State:= STATE_CLOSE;
							m_ConnectionWatchdog(IN:=FALSE);(*reset connection watchdog*)
							diError := 16#8009;
						END_IF
					0:(* socket was "gracefully closed"  *)
						m_State:= STATE_CLOSE;
						diError := 16#8003;
					ELSE
						(* Copy received data into receive buffer *)
						(********************************)
						FOR i:= 0 TO DINT_TO_INT(m_BytesReceived	)-1 DO
							aReceiveBuffer[diReceiveCount]:= m_ReceiveBuffer[i];
							diReceiveCount:=(diReceiveCount+1) MOD SIZEOF(aReceiveBuffer);
						END_FOR

						m_ConnectionWatchdog(IN:=FALSE);(*reset connection watchdog*)
					END_CASE

				(*send data*)
				IF xStartSend	 THEN
					m_State := STATE_TX;
				END_IF

	STATE_TX:	 (* send TCP-message *)
		m_diReturn := SysSockSend(diSocket := m_Socket,
								  pbyBuffer := ADR(ptSendData^[m_count]),(*geändert V1.4 bisher: [0] *)
								  diBufferSize := diSendCount-m_count,
								  diFlags :=m_Flags);
		CASE m_diReturn OF
		-1:	(* ERROR or data could not yet be send (V1.3 due to new FW11) *)
			m_ConnectionWatchdog(IN:=TRUE , PT:=tServerTimeOut );
			IF m_connectionWatchdog.Q THEN
				m_State:= STATE_CLOSE;
				m_ConnectionWatchdog(IN:=FALSE);(*reset connection watchdog*)
				diError := 16#8007;
			END_IF
		0: (* socket was "gracefully closed"  *)
			m_State := STATE_CLOSE;
			diError := 16#8003;
		ELSE (* succesful *)
			m_count:=m_count+m_diReturn;
			IF m_count>=diSendCount THEN
				diError := 16#0000;
				m_State := STATE_RX;
				m_count:=0;
				xStartSend:=FALSE;
			END_IF
			m_ConnectionWatchdog(IN:=FALSE);(*reset connection watchdog*)
		END_CASE


		STATE_CLOSE:	(* Close the server *)

		IF ADR(%MW0)=16#30000000  OR ADR(%MW0)=16#20000000 THEN (*841 or 881*)
			;
		ELSE
			IF m_Socket>=0 THEN
				SysSockShutdown(m_Socket, 0);;(*870*)
			END_IF
		END_IF
		IF m_Socket>=0 THEN
			SysSockClose( m_Socket);
		END_IF
		xClientConnected:= FALSE;
		m_State:= STATE_OPEN; (* Try to open the server again *)
		m_ConnectionWatchdog(IN:=FALSE);(*reset connection watchdog*)

		STATE_ERROR_TRAP: (* Error Read/Write socket  *)
			m_State:= STATE_ERROR_TRAP;

	ELSE  (* Bad FSM code trap  *)
			m_State:= STATE_ERROR_TRAP;
			diError:= 16#8008;
	END_CASE;
ELSE
	IF m_State <> STATE_INIT THEN
		IF ADR(%MW0)=16#30000000  OR ADR(%MW0)=16#20000000 THEN (*841 or 881*)
			;
		ELSE
			IF m_Socket>=0 THEN
				SysSockShutdown(m_Socket, 0);;(*870*)
			END_IF
		END_IF
		IF m_Socket>=0 THEN
			SysSockClose( m_Socket);
		END_IF
		IF ADR(%MW0)=16#30000000  OR ADR(%MW0)=16#20000000 THEN (*841 or 881*)
			;
		ELSE
			IF m_ServerSocket>=0 THEN
				SysSockShutdown(m_ServerSocket, 0);;(*870*)
			END_IF
		END_IF
		IF m_ServerSocket>=0 THEN
			SysSockClose( m_ServerSocket);
		END_IF
		xClientConnected:= FALSE;
		diError:= 0;
		m_State:= STATE_init; (* Try to open the server again *)
		m_ConnectionWatchdog(IN:=FALSE);(*reset connection watchdog*)
	END_IF
END_IF
END_FUNCTION_BLOCK

(* POU Utils Functions/HEXTORAW, ST *)
FUNCTION HEXTORAW : WORD
VAR_INPUT
	pString		: POINTER TO BYTE;
	StringLen	: WORD;
	pData		: POINTER TO BYTE;
END_VAR
VAR
	xl: WORD;
	xi: WORD;
	xr: BYTE;
END_VAR
xl:=0;
xi:=0;

WHILE xi<StringLen DO

	IF pString^>=97 AND pString^<=102 THEN
		xr := pString^ - 87;
	ELSIF pString^>=65 AND pString^<=70 THEN
		xr := pString^ - 55;
	ELSIF pString^>=48 AND pString^<=57 THEN
		xr := pString^ - 48;
	ELSE
		xr := 16;
	END_IF

	IF xr<16 THEN
		IF (xi AND 1)=0 THEN
			pData^ := xr * 16;
		ELSE
			pData^ := pData^ + xr;
			pData := pData + 1;
			xl := xl + 1;
		END_IF
	END_IF

	xi := xi + 1;
	pString := pString + 1;

END_WHILE

HEXTORAW:=xl;
END_FUNCTION

(* POU Utils Functions/RAWTOHEX, ST *)
FUNCTION RAWTOHEX : WORD
VAR_INPUT
	pData: POINTER TO BYTE;
	DataLen: WORD;
	pString: POINTER TO BYTE;
END_VAR
VAR
	xl: WORD;
END_VAR
xl:=0;

WHILE DataLen>0 DO

	pString^ := (pData^ / 16#10) + 48 + (((pData^ / 16#10)/10)*7);
	pString:=pString+1;
	pString^ := (pData^ AND 16#0F)  + 48 + (((pData^ AND 16#0F)/10)*7);
	pString:=pString+1;
	pData:=pData+1;
	DataLen:=DataLen-1;
	xl:=xl+2;

END_WHILE

(*pString^:=0;*)

RAWTOHEX:=xl;
END_FUNCTION

(* POU Utils/USRLED_Update, ST *)
PROGRAM USRLED_Update
VAR
	OldStatus: en_SYS_Status;

	aFS : ARRAY [0..24] OF FLASHING_SEQUENCE :=
		(Colour:=GREEN,  Frequency:=1,   Relation:=128, Duration:=t#0s,    NextIndex:=0),  (* 0 => RUNNING *)
		(Colour:=ORANGE, Frequency:=1,   Relation:=128, Duration:=t#0s,    NextIndex:=1),  (* 1 => INIT *)
		(Colour:=RED,    Frequency:=4,   Relation:=128, Duration:=t#0s,    NextIndex:=2),  (* 2 => ERROR *)
		(Colour:=RED,    Frequency:=10,  Relation:=128, Duration:=t#0s,    NextIndex:=3),  (* 3 => ALARM *)
		(Colour:=ORANGE, Frequency:=200, Relation:=16,  Duration:=t#100ms, NextIndex:=11), (* 10 *)
		(Colour:=ORANGE, Frequency:=200, Relation:=32,  Duration:=t#100ms, NextIndex:=12),
		(Colour:=ORANGE, Frequency:=200, Relation:=64,  Duration:=t#100ms, NextIndex:=13),
		(Colour:=ORANGE, Frequency:=200, Relation:=128, Duration:=t#100ms, NextIndex:=14),
		(Colour:=ORANGE, Frequency:=200, Relation:=192, Duration:=t#100ms, NextIndex:=15),
		(Colour:=ORANGE, Frequency:=200, Relation:=128, Duration:=t#100ms, NextIndex:=16),
		(Colour:=ORANGE, Frequency:=200, Relation:=64,  Duration:=t#100ms, NextIndex:=17),
		(Colour:=ORANGE, Frequency:=200, Relation:=32,  Duration:=t#100ms, NextIndex:=18),
		(Colour:=ORANGE, Frequency:=200, Relation:=16,  Duration:=t#100ms, NextIndex:=19),
		(Colour:=ORANGE, Frequency:=200, Relation:=8,   Duration:=t#100ms, NextIndex:=10),
		(Colour:=GREEN,  Frequency:=200, Relation:=16,  Duration:=t#100ms, NextIndex:=21), (* 20 *)
		(Colour:=GREEN,  Frequency:=200, Relation:=32,  Duration:=t#100ms, NextIndex:=22),
		(Colour:=GREEN,  Frequency:=200, Relation:=64,  Duration:=t#100ms, NextIndex:=23),
		(Colour:=GREEN,  Frequency:=200, Relation:=128, Duration:=t#100ms, NextIndex:=24),
		(Colour:=GREEN,  Frequency:=200, Relation:=192, Duration:=t#100ms, NextIndex:=25),
		(Colour:=GREEN,  Frequency:=200, Relation:=128, Duration:=t#100ms, NextIndex:=26),
		(Colour:=GREEN,  Frequency:=200, Relation:=64,  Duration:=t#100ms, NextIndex:=27),
		(Colour:=GREEN,  Frequency:=200, Relation:=32,  Duration:=t#100ms, NextIndex:=28),
		(Colour:=GREEN,  Frequency:=200, Relation:=16,  Duration:=t#100ms, NextIndex:=29),
		(Colour:=GREEN,  Frequency:=200, Relation:=8,   Duration:=t#100ms, NextIndex:=20);

	pFS : POINTER TO FLASHING_SEQUENCE;


END_VAR
IF Sys.Status <> OldStatus THEN

	OldStatus:=Sys.Status;

	CASE OldStatus OF

		S_STARTUP:
			pFS:=ADR(aFS);
			SET_FLASHING_SEQUENCE(EN:=TRUE, POINTER_TO_POINTER_TO_ARRAY:=ADR(pFS));
			SET_FLASHING_SEQUENCE_INDEX(EN:=TRUE, IMMEDIATE:=FALSE, INDEX:=1);
			START_FLASHING_SEQUENCE(EN:=TRUE);

		S_RUNNING:
			SET_FLASHING_SEQUENCE_INDEX(EN:=TRUE, IMMEDIATE:=TRUE, INDEX:=0);

	END_CASE

END_IF
END_PROGRAM

(* POU Plant/SYS_Proc, ST *)
PROGRAM SYS_Proc
VAR
(*	fALARM_PB		:FLT_TAP;
	fALARM_TB		:FLT_TAP;
	fALARM_PM		:FLT_TAP; *)

(*	fGZB_ST			:FLT_TAP; (* GATEWAY ZIGBEE *)*)
(*	fVPN_OUT1		:FLT_TAP; (* VPN - CONNECT *)*)
	fVPN_OUT2		:FLT_TAP; (* VPN - STATUS *)
(*	fKEY_CT_ST		:FLT_TAP; (* DOOR01 - Porta primaria *)*)
(*	fKEY_SCT_ST		:FLT_TAP; (* DOOR02 - Porta secondaria *)*)
	fKEY_QE_ST		:FLT_TAP; (* DOOR03 - Quadro Elettrico *)

END_VAR
(*************** ISPESL *****************)
(*
fALARM_PB(IN:=ALARM_PB);
IF fALARM_PB.EVH THEN
	LogEv(EL_AlarmStop,EO_PBV,1,1,'Over_Pressure_Alarm');
END_IF

fALARM_TB(IN:=ALARM_TB);
IF fALARM_TB.EVH THEN
	LogEv(EL_AlarmStop,EO_TBV,1,1,'Over_Temperature_Alarm');
END_IF

fALARM_PM(IN:=ALARM_PM);
IF fALARM_PM.EVH THEN
	LogEv(EL_AlarmStop,EO_PMV,1,1,'Under_Pressure_Alarm');
END_IF
*)
(****************************************)

(*### VPN Connection Check ###*)(*
fVPN_OUT1(IN:=VPN_OUT1);
IF fVPN_OUT1.EVH THEN
	LogEv(EL_Log,EO_VPN,1,1,'CONNECT_ON');
END_IF
IF fVPN_OUT1.EVL THEN
	LogEv(EL_Log,EO_VPN,1,2,'CONNECT_OFF');
END_IF*)

(*### VPN Status Check ###*)
fVPN_OUT2(IN:=VPN_OUT2);
IF fVPN_OUT2.EVH THEN
	LogEv(EL_Log,EO_VPN,1,3,'STATUS_UP');
END_IF
IF fVPN_OUT2.EVL THEN
	LogEv(EL_Wrn,EO_VPN,1,4,'STATUS_DOWN');
END_IF

(*### DOOR01 Status Check ###*)(*
fKEY_CT_ST(IN:=KEY_CT_ST);
IF fKEY_CT_ST.EVH THEN
	LogEv(EL_Log,EO_DOOR,1,2,'Centrale_termica_Close');
END_IF
IF fKEY_CT_ST.EVL THEN
	LogEv(EL_Wrn,EO_DOOR,1,1,'Centrale_termica_Open');
END_IF*)

(*### DOOR02 Status Check ###*)(*
fKEY_SCT_ST(IN:=KEY_SCT_ST);
IF fKEY_SCT_ST.EVH THEN
	LogEv(EL_Log,EO_DOOR,2,2,'Sottocentrale_termica_Close');
END_IF
IF fKEY_SCT_ST.EVL THEN
	LogEv(EL_Wrn,EO_DOOR,2,1,'Sottocentrale_termica_Open');
END_IF*)

(*### DOOR03 Status Check ###*)
fKEY_QE_ST(IN:=KEY_QE_ST);
IF fKEY_QE_ST.EVH THEN
	LogEv(EL_Log,EO_DOOR,3,2,'Quadro_Close');
END_IF
IF fKEY_QE_ST.EVL THEN
	LogEv(EL_Wrn,EO_DOOR,3,1,'Quadro_Open');
END_IF
END_PROGRAM

(* POU Utils Functions/FLT_TAP, ST *)
FUNCTION_BLOCK FLT_TAP
VAR_INPUT
	IN		: BOOL;
	TAP		: BYTE:=4;
	INITEV	: BOOL:=TRUE;
END_VAR
VAR_OUTPUT
	OUT		: BOOL;
	EVH		: BOOL;
	EVL		: BOOL;
END_VAR
VAR
	init	: BOOL:=FALSE;
	cnt		: BYTE;
END_VAR
EVH:=FALSE;
EVL:=FALSE;

IF NOT init THEN
	init := TRUE;
	IF INITEV THEN
		OUT  := NOT IN;
		cnt  := TAP;
	ELSE
		OUT  := IN;
	END_IF
END_IF

IF OUT<>IN THEN
	cnt:=cnt+1;
	IF cnt>TAP THEN
		OUT:=IN;
		cnt:=0;
		IF OUT THEN EVH:=TRUE; ELSE EVL:=TRUE; END_IF
	END_IF
ELSE
	cnt:=0;
END_IF
END_FUNCTION_BLOCK

(* POU TCP_Logger/LogEv, ST *)
FUNCTION LogEv : BOOL
VAR_INPUT
	Level	: en_Logger_ErrLev;
	Object  : en_SYS_Objects;
	Index	: WORD;
	Error	: WORD;
	Message : STRING;
END_VAR
VAR
	s1 : STRING(160);
	i  : INT;
END_VAR
(* Execute error level operations *)
CASE Level OF
	EL_Wrn: 		Sys.Warning:=TRUE;
	EL_Alarm: 		Sys.Alarm  :=TRUE;
	EL_AlarmStop: 	Sys.Alarm  :=TRUE; (* GO TO STOP STATE!! *)
END_CASE

(* Fill lastlog list *)
s1:=CONCAT(Sys.Time_LogString,';Lev=');
s1:=CONCAT(s1,INT_TO_STRING(Level));
s1:=CONCAT(s1,';Obj=');
s1:=CONCAT(s1,INT_TO_STRING(Object));
s1:=CONCAT(s1,';Idx=');
s1:=CONCAT(s1,WORD_TO_STRING(Index));
s1:=CONCAT(s1,';Err=');
s1:=CONCAT(s1,WORD_TO_STRING(Error));
Sys.LastLogs_Dat[Sys.LastLogs_Idx]:=s1;
Sys.LastLogs_Msg[Sys.LastLogs_Idx]:=Message;
Sys.LastLogs_Idx:=Sys.LastLogs_Idx+1;
IF Sys.LastLogs_Idx>5 THEN Sys.LastLogs_Idx:=0; END_IF

(*---------------------------------------------------------------*)
	Logger_Head();
(*---------------------------------------------------------------*)

(* Insert ERR *)
s1:=CONCAT('&ERR=',INT_TO_STRING(Level));
s1:=CONCAT(s1,';');
s1:=CONCAT(s1,INT_TO_STRING(Object));
s1:=CONCAT(s1,';');
s1:=CONCAT(s1,WORD_TO_STRING(Index));
s1:=CONCAT(s1,';');
s1:=CONCAT(s1,WORD_TO_STRING(Error));
s1:=CONCAT(s1,';');
ADDSTRING(ADR(Logger.TData), ADR(s1), Logger.TLen);
s1:=Message;
STR_NOSPACES(ADR(s1));
ADDSTRING(ADR(Logger.TData), ADR(s1), Logger.TLen);

(*---------------------------------------------------------------*)
	Logger_Send();
(*---------------------------------------------------------------*)
END_FUNCTION

(* POU TCP_Logger/Logger_Head, ST *)
FUNCTION Logger_Head : BOOL
VAR
	s1 : STRING(160);
	i  : BYTE;
END_VAR
Logger.TLen:=0;
(* Set GET header *)
ADDSTRING(ADR(Logger.TData), ADR(Logger_GETSTART), Logger.TLen);

(* Insert Header *)
s1:=INSERT('ID=&V=1&D=',DWORD_TO_STRING(Plant_SN),3);
s1:=CONCAT(s1,Sys.Time_LogString);
s1:=CONCAT(s1,'&S=');
IF Sys.Alarm THEN i:=2; ELSIF Sys.Warning THEN i:=1; ELSE i:=0; END_IF
s1:=CONCAT(s1,BYTE_TO_STRING(i));
ADDSTRING(ADR(Logger.TData), ADR(s1), Logger.TLen);
END_FUNCTION

(* POU Utils Functions/ADDSTRING, ST *)
FUNCTION ADDSTRING : BOOL (* Append string to a byte buffer *)
VAR_INPUT
	pTxData: POINTER TO BYTE;
	pString: POINTER TO BYTE;
END_VAR
VAR_IN_OUT
	TxLen: DINT;
END_VAR
VAR
END_VAR
pTxData:=pTxData+TxLen;
WHILE pString^<>0 DO
	pTxData^:=pString^;
	pString:=pString+1;
	pTxData:=pTxData+1;
	TxLen:=TxLen+1;
END_WHILE
END_FUNCTION

(* POU Utils Functions/STR_NOSPACES, ST *)
FUNCTION STR_NOSPACES : BOOL (* Replace spaces and bad chars with allowed ones, used as HTTP-GET validator *)
VAR_INPUT
	pString: POINTER TO BYTE;
END_VAR
VAR
END_VAR
WHILE pString^<>0 DO
	IF pString^=16#20 (* space *) THEN pString^:=16#5F; (*'_'*) END_IF
	pString:=pString+1;
END_WHILE
END_FUNCTION

(* POU TCP_Logger/Logger_Send, ST *)
FUNCTION Logger_Send : BOOL
VAR
	hFile: 	DWORD;
	pos:	DWORD;
END_VAR
(* Finalize string *)
ADDSTRING(ADR(Logger.TData), ADR(Logger_GETEND), Logger.TLen);

(* Read log position *)
pos:=SysFileGetSize(Logger_DataFile);
(* Check log size, bckup and erase if no pending messages *)
IF pos>10000000 (*10M*) THEN
	hFile:=SysFileOpen(Logger_IndexFile,'r');
	IF hFile=0 THEN
		SysFileDelete(Logger_DataFileOld);
		SysFileRename(Logger_DataFile,Logger_DataFileOld);
		pos:=0;
	ELSE
		SysFileClose(hFile);
	END_IF
END_IF
(* Write message on log file *)
hFile:=SysFileOpen(Logger_DataFile,'a');
IF hFile<>0 THEN
	SysFileWrite(hFile, ADR(Logger.TData), Logger.TLen);
	SysFileClose(hFile);
ELSE
	Sys.Warning:=TRUE;
END_IF


(* Check logger status *)
IF Logger.SendReq=FALSE THEN
	(* Set log position for recovery *)
	Logger.SendIdx:=pos;
	(* Copy message data *)
	MEMCPY(ADR(Logger.TData),ADR(Logger.SendData),DINT_TO_WORD(Logger.TLen));
	Logger.SendLen:=Logger.TLen;
	(* Trigger request *)
	Logger.SendReq:=TRUE;
ELSE
	(* Add message position+size in recovery indexes *)
	hFile:=SysFileOpen(Logger_IndexFile,'a');
	SysFileWrite(hFile, ADR(pos), SIZEOF(pos));
	SysFileWrite(hFile, ADR(Logger.TLen), SIZEOF(Logger.TLen));
	SysFileClose(hFile);
END_IF
END_FUNCTION

(* POU Utils Functions/MEMCPY, ST *)
FUNCTION MEMCPY:BOOL
VAR_INPUT
	pSourceAddress:POINTER TO ARRAY[1..2] OF BYTE;
	pDestinationAddress:POINTER TO ARRAY[1..2] OF BYTE;
	BytesToCopy:WORD;
END_VAR
VAR
END_VAR
WHILE (BytesToCopy > 0) DO
	pDestinationAddress^[1]:=pSourceAddress^[1]; (* copy bytes from source to destination *)
	pDestinationAddress:=ADR(pDestinationAddress^[2]); (* increment destination *)
	pSourceAddress:=ADR(pSourceAddress^[2]);(* increment source *)
	BytesToCopy:=BytesToCopy -1; (* decrement number of bytes to copy *)
END_WHILE
END_FUNCTION

(* POU Utils Functions/AVERAGE_T, ST *)
FUNCTION_BLOCK AVERAGE_T
VAR_INPUT
	IN: 	INT;
END_VAR
VAR_OUTPUT
	HI:		INT;
	AVG:	INT;
	LOW:	INT;
	ERR:	BOOL;
END_VAR
VAR
	sum:	DINT;
	cnt:	WORD;
END_VAR
IF cnt>=65000 THEN
	ERR:=TRUE;
	Read();
	sum := sum - AVG;
	cnt := cnt + 1;
END_IF

sum := sum + IN;
cnt := cnt + 1;

IF IN<LOW THEN  LOW:=IN; END_IF
IF IN>HI  THEN HI :=IN; END_IF
END_FUNCTION_BLOCK
ACTION Read:
AVG := DINT_TO_INT(sum/cnt);
END_ACTION
ACTION Reset:
HI:=IN;
AVG:=IN;
LOW:=IN;
ERR:=FALSE;

sum:=IN;
cnt:=1;
END_ACTION

(* POU Utils Functions/COPY_32SWAP16, ST *)
FUNCTION COPY_32SWAP16:BOOL
VAR_INPUT
	pSourceAddress		:POINTER TO ARRAY[1..2] OF WORD;
	pDestinationAddress	:POINTER TO ARRAY[1..2] OF WORD;
END_VAR
VAR
END_VAR
pDestinationAddress^[1]:=pSourceAddress^[2];
pDestinationAddress^[2]:=pSourceAddress^[1];
END_FUNCTION

(* POU Utils/CSV_Log, ST *)
FUNCTION CSV_Log : BOOL
VAR_INPUT
END_VAR
VAR CONSTANT
	LogFileName:STRING:='S:\LOGS_ID2V3.CSV';
END_VAR
VAR
	s1 : STRING(256);
	hFile: 	DWORD;
END_VAR
(* Check file presence *)
hFile:=SysFileOpen(LogFileName,'r');
IF hFile=0 THEN
	(*** File not exist *** Create file and write header *)
	hFile:=SysFileOpen(LogFileName,'w');
	IF hFile<>0 THEN
		(* Write CSV header *)
		s1:='DATE-TIME;T-Amb;T-GRU01-SetP;T-GRU01-Send;T-GRU01-Ret;T-GRU01-Amb;T_S01;T_S02;F-PDC01-Flow;T-PDC01-Send;T-PDC01-Ret;';
		SysFileWrite(hFile, ADR(s1), LEN(s1));
		s1:='T-CTB01-Send;T-CTB01-Ret;F-CTB01-Flow;P-CTB01-Power;E-CTB01-Energy';
		SysFileWrite(hFile, ADR(s1), LEN(s1));
		SysFileWrite(hFile, ADR(Logger_CRLF), LEN(Logger_CRLF));
	END_IF
ELSE
	(*** File exist *** Close file and reopen in append mode *)
	SysFileClose(hFile);
	hFile:=SysFileOpen(LogFileName,'a');
END_IF

(* Log to file *)
IF hFile<>0 THEN
	(* Date stamp *)
	s1:=REPLACE( Sys.Time_LogString , ' ' , 1 , 11 );
	SysFileWrite(hFile, ADR(s1), LEN(s1));
	(* Log data 1 *)
	s1:=CONCAT(';', INT_TO_STRING(T_AMB) );
	s1:=CONCAT(s1 , ';');
	s1:=CONCAT(s1 , INT_TO_STRING(GRU01.ActSetPoint) );
	s1:=CONCAT(s1 , ';');
	s1:=CONCAT(s1 , INT_TO_STRING(GRU01.TSend) );
	s1:=CONCAT(s1 , ';');
	s1:=CONCAT(s1 , INT_TO_STRING(GRU01.TRet) );
	s1:=CONCAT(s1 , ';');
	s1:=CONCAT(s1 , INT_TO_STRING(GRU01.TAmb) );
	s1:=CONCAT(s1 , ';');
	s1:=CONCAT(s1 , INT_TO_STRING(T_S01) );
	s1:=CONCAT(s1 , ';' );
	s1:=CONCAT(s1 , INT_TO_STRING(T_S02) );
	s1:=CONCAT(s1 , ';' );
	s1:=CONCAT(s1 , WORD_TO_STRING(PDC01.Flow) );
	s1:=CONCAT(s1 , ';' );
	s1:=CONCAT(s1 , INT_TO_STRING(PDC01.TSend) );
	s1:=CONCAT(s1 , ';');
	s1:=CONCAT(s1 , INT_TO_STRING(PDC01.TRet) );
	SysFileWrite(hFile, ADR(s1), LEN(s1));
	(* Log data 2 *)
	s1:=CONCAT(';', CTB01.M1.utFTemp.Value );
	s1:=CONCAT(s1 , ';');
	s1:=CONCAT(s1 , CTB01.M1.utRTemp.Value );
	s1:=CONCAT(s1 , ';');
	s1:=CONCAT(s1 , CTB01.M1.utFlow.Value );
	s1:=CONCAT(s1 , ';');
	s1:=CONCAT(s1 , CTB01.M1.utPower.Value );
	s1:=CONCAT(s1 , ';');
	s1:=CONCAT(s1 , CTB01.M1.utEnergy.Value );
	SysFileWrite(hFile, ADR(s1), LEN(s1));
	(* Add line CRLF and close *)
	SysFileWrite(hFile, ADR(Logger_CRLF), LEN(Logger_CRLF));
	SysFileClose(hFile);
END_IF
END_FUNCTION

(* POU Utils Functions/FLT_EVENT, ST *)
FUNCTION_BLOCK FLT_EVENT
VAR_INPUT
	IN		: BOOL;
	INITEV	: BOOL:=TRUE;
END_VAR
VAR_OUTPUT
	EVH		: BOOL;
	EVL		: BOOL;
END_VAR
VAR
	init	: BOOL:=FALSE;
	old		: BOOL;
END_VAR
EVH:=FALSE;
EVL:=FALSE;

IF NOT init THEN
	init:=TRUE;
	IF INITEV THEN
		old := NOT IN;
	ELSE
		old := IN;
	END_IF
END_IF

IF old<>IN THEN
	old:=IN;
	IF IN THEN EVH:=TRUE; ELSE EVL:=TRUE; END_IF
END_IF
END_FUNCTION_BLOCK

(* POU Utils Functions/FLT_TIME, ST *)
FUNCTION_BLOCK FLT_TIME
VAR_INPUT
	IN		: BOOL;
	TTAP	: TIME:=T#5s;
	INITEV	: BOOL:=TRUE;
END_VAR
VAR_OUTPUT
	OUT		: BOOL;
	EVH		: BOOL;
	EVL		: BOOL;
END_VAR
VAR
	init	: BOOL:=FALSE;
	timer	: TON;
END_VAR
EVH:=FALSE;
EVL:=FALSE;

IF NOT init THEN
	init := TRUE;
	IF INITEV THEN
		OUT  := NOT IN;
	ELSE
		OUT  := IN;
	END_IF
END_IF

IF OUT<>IN THEN
	timer(IN:=TRUE,PT:=TTAP);
	IF timer.Q THEN
		OUT:=IN;
		timer(IN:=FALSE);
		IF OUT THEN EVH:=TRUE; ELSE EVL:=TRUE; END_IF
	END_IF
ELSE
	timer(IN:=FALSE);
END_IF
END_FUNCTION_BLOCK

(* POU TCP_Logger/LogTrig, ST *)
FUNCTION LogTrig : BOOL
VAR
	s1 : STRING(160);
	i  : BYTE;
END_VAR
(*---------------------------------------------------------------*)
	Logger_Head();
(*---------------------------------------------------------------*)


(* Insert TPVs *)
s1:=CONCAT('&TPV=',INT_TO_STRING(T_S01));
s1:=CONCAT(s1,';'); s1:=CONCAT(s1,INT_TO_STRING(T_S02));
s1:=CONCAT(s1,';'); s1:=CONCAT(s1,INT_TO_STRING(GRU01.TSend));
s1:=CONCAT(s1,';'); s1:=CONCAT(s1,INT_TO_STRING(GRU01.TRet));
s1:=CONCAT(s1,';'); s1:=CONCAT(s1,INT_TO_STRING(GRU01.TAmb));
ADDSTRING(ADR(Logger.TData), ADR(s1), Logger.TLen);

(* Insert GRU01 *)
s1:=CONCAT('&GRU01=',INT_TO_STRING(GRU01.ActSetPoint));
s1:=CONCAT(s1,';'); s1:=CONCAT(s1,INT_TO_STRING(0));
s1:=CONCAT(s1,';'); s1:=CONCAT(s1,BYTE_TO_STRING(GRU01.Status_Log));
ADDSTRING(ADR(Logger.TData), ADR(s1), Logger.TLen);
(* Insert PDC01 *)
s1:=CONCAT('&PDC01=',INT_TO_STRING(0));
s1:=CONCAT(s1,';'); s1:=CONCAT(s1,WORD_TO_STRING(PDC01.Power/100));
s1:=CONCAT(s1,';'); s1:=CONCAT(s1,BYTE_TO_STRING(PDC01.Status_Log));
ADDSTRING(ADR(Logger.TData), ADR(s1), Logger.TLen);
(* Insert CAL01 *)
s1:=CONCAT('&CAL01=',INT_TO_STRING(0));
s1:=CONCAT(s1,';'); s1:=CONCAT(s1,WORD_TO_STRING(100*CAL01.OnOff));
s1:=CONCAT(s1,';'); s1:=CONCAT(s1,BYTE_TO_STRING(CAL01.Status_Log));
ADDSTRING(ADR(Logger.TData), ADR(s1), Logger.TLen);
(* Insert CAL02 *)
s1:=CONCAT('&CAL02=',INT_TO_STRING(0));
s1:=CONCAT(s1,';'); s1:=CONCAT(s1,WORD_TO_STRING(100*CAL02.OnOff));
s1:=CONCAT(s1,';'); s1:=CONCAT(s1,BYTE_TO_STRING(CAL02.Status_Log));
ADDSTRING(ADR(Logger.TData), ADR(s1), Logger.TLen);

(* Insert CIR01 *)
s1:=CONCAT('&CIR01=',SEL(CIR01.CIR_EN,'0','100'));
s1:=CONCAT(s1,';'); s1:=CONCAT(s1,BYTE_TO_STRING(CIR01.Status_Log));
ADDSTRING(ADR(Logger.TData), ADR(s1), Logger.TLen);
(* Insert CIR02 *)
s1:=CONCAT('&CIR02=',SEL(CIR02.CIR_EN,'0','100'));
s1:=CONCAT(s1,';'); s1:=CONCAT(s1,BYTE_TO_STRING(CIR02.Status_Log));
ADDSTRING(ADR(Logger.TData), ADR(s1), Logger.TLen);
(* Insert CIR03 *)
s1:=CONCAT('&CIR03=',SEL(CIR03.CIR_EN,'0','100'));
s1:=CONCAT(s1,';'); s1:=CONCAT(s1,BYTE_TO_STRING(CIR03.Status_Log));
ADDSTRING(ADR(Logger.TData), ADR(s1), Logger.TLen);
(* Insert CIR04 *)
s1:=CONCAT('&CIR04=',SEL(CIR04.CIR_EN,'0','100'));
s1:=CONCAT(s1,';'); s1:=CONCAT(s1,BYTE_TO_STRING(CIR04.Status_Log));
ADDSTRING(ADR(Logger.TData), ADR(s1), Logger.TLen);
(* Insert CIR05 *)
s1:=CONCAT('&CIR05=',SEL(CIR05.CIR_EN,'0','100'));
s1:=CONCAT(s1,';'); s1:=CONCAT(s1,BYTE_TO_STRING(CIR05.Status_Log));
ADDSTRING(ADR(Logger.TData), ADR(s1), Logger.TLen);
(* Insert CIR06 *)
s1:=CONCAT('&CIR06=',SEL(CIR06.CIR_EN,'0','100'));
s1:=CONCAT(s1,';'); s1:=CONCAT(s1,BYTE_TO_STRING(CIR06.Status_Log));
ADDSTRING(ADR(Logger.TData), ADR(s1), Logger.TLen);

(* Insert CRON01 *)
s1:=CONCAT('&CRON01=',INT_TO_STRING(CRON01.SetPoint));
s1:=CONCAT(s1,';'); s1:=CONCAT(s1,BYTE_TO_STRING(CRON01.Status_Log));
ADDSTRING(ADR(Logger.TData), ADR(s1), Logger.TLen);
(* Insert CRON02 *)
s1:=CONCAT('&CRON02=',INT_TO_STRING(CRON02.SetPoint));
s1:=CONCAT(s1,';'); s1:=CONCAT(s1,BYTE_TO_STRING(CRON02.Status_Log));
ADDSTRING(ADR(Logger.TData), ADR(s1), Logger.TLen);
(* Insert CRON03 *)
s1:=CONCAT('&CRON03=',INT_TO_STRING(CRON03.SetPoint));
s1:=CONCAT(s1,';'); s1:=CONCAT(s1,BYTE_TO_STRING(CRON03.Status_Log));
ADDSTRING(ADR(Logger.TData), ADR(s1), Logger.TLen);
(* Insert CRON04 *)
s1:=CONCAT('&CRON04=',INT_TO_STRING(CRON04.SetPoint));
s1:=CONCAT(s1,';'); s1:=CONCAT(s1,BYTE_TO_STRING(CRON04.Status_Log));
ADDSTRING(ADR(Logger.TData), ADR(s1), Logger.TLen);
(* Insert CRON05 *)
s1:=CONCAT('&CRON05=',INT_TO_STRING(CRON05.SetPoint));
s1:=CONCAT(s1,';'); s1:=CONCAT(s1,BYTE_TO_STRING(CRON05.Status_Log));
ADDSTRING(ADR(Logger.TData), ADR(s1), Logger.TLen);
(* Insert CRON06 *)
s1:=CONCAT('&CRON06=',INT_TO_STRING(CRON06.SetPoint));
s1:=CONCAT(s1,';'); s1:=CONCAT(s1,BYTE_TO_STRING(CRON06.Status_Log));
ADDSTRING(ADR(Logger.TData), ADR(s1), Logger.TLen);

(* Insert CTL01 *)
s1:=CONCAT('&CTL01=',DWORD_TO_STRING(CTL01_Count));
s1:=CONCAT(s1,';'); s1:=CONCAT(s1,BYTE_TO_STRING(CTL01.Status_Log));
ADDSTRING(ADR(Logger.TData), ADR(s1), Logger.TLen);

(* Insert CTB01 *)
s1:=CONCAT('&CTB01=',CTB01.M1.utFTemp.Value);
s1:=CONCAT(s1,';'); s1:=CONCAT(s1 , CTB01.M1.utRTemp.Value );
s1:=CONCAT(s1,';'); s1:=CONCAT(s1 , CTB01.M1.utFlow.Value );
s1:=CONCAT(s1,';'); s1:=CONCAT(s1 , CTB01.M1.utPower.Value );
s1:=CONCAT(s1,';'); s1:=CONCAT(s1 , CTB01.M1.utEnergy.Value );
s1:=CONCAT(s1,';'); s1:=CONCAT(s1 , BYTE_TO_STRING(CTB01.Status_Log) );
ADDSTRING(ADR(Logger.TData), ADR(s1), Logger.TLen);


(*---------------------------------------------------------------*)
	Logger_Send();
(*---------------------------------------------------------------*)
END_FUNCTION

(* POU Utils Functions/MEMCLR, ST *)
FUNCTION MEMCLR:BOOL
VAR_INPUT
	pDestinationAddress:POINTER TO ARRAY[1..2] OF BYTE;
	BytesToClear:WORD;
END_VAR
VAR
END_VAR
WHILE (BytesToClear > 0) DO
	pDestinationAddress^[1]:=0;
	pDestinationAddress:=ADR(pDestinationAddress^[2]); (* increment destination *)
	BytesToClear:=BytesToClear -1; (* decrement number of bytes to copy *)
END_WHILE
END_FUNCTION

(* POU Plant_Objects/obj_CAL_ROBUR_AY, ST *)
FUNCTION_BLOCK obj_CAL_ROBUR_AY
(* === CALDAIA ROBUR AY from DDC ===
   v1.0[16/04/15] - Versioning
*)
VAR_INPUT
	(* Settings *)
	ID				: BYTE; (* Index of instanced object *)
	NetID			: WORD; (* Network ID on ROBUR DDC *)

	(* Controls *)
	Rearm			: BOOL; (* 40244=UID(u16-Unit), 40245=1(u16-Reset) *)

	(* States *)
	OnOff			: WORD; (* 12028 + 0*64 *)
	TSend			: INT;	(* 35023 + 0*250 *)
	TRet			: INT;	(* 35024 + 0*250 *)
	Power			: WORD; (* 35044 + 0*250 = Power feedback percentage 0-100% *)
	Status			: WORD; (* 35061 + 0*250 = General alarm bits1&0 00:OK 01:LOG 10:WRN 11:ERR *)

END_VAR
VAR_OUTPUT
	(* Visu/Log *)
	Status_Log		: BYTE;
	Status_Vis : DWORD;
END_VAR
VAR
END_VAR
(* Status color *)
   IF (Status AND 16#3)=16#3 THEN Status_Log:=2; Status_Vis:=COLOR_RED;
ELSIF (Status AND 16#3)>1    THEN Status_Log:=1; Status_Vis:=COLOR_YELLOW;
              				 ELSE Status_Log:=0; Status_Vis:=SEL(OnOff=1,COLOR_GREEN_OFF,COLOR_GREEN);
END_IF
END_FUNCTION_BLOCK

(* POU Plant_Objects/obj_CIR, ST *)
FUNCTION_BLOCK obj_CIR
(* === CIRCOLATORE STANDARD ===
   v1.0[16/04/15] - Versioning
*)
VAR_INPUT
	(* Settings *)
	ID				: BYTE;
	Chk_CntTrig		: BYTE:=10;	(* Check error trigger 5s *)
	(* Controls *)
	Ctrl_SetPoint 	: INT;
(*	CIR_RUN			: BOOL; (* Standard run request *) *)
	CIR_RUN_REQ		: BOOL; (* External run request (no heat or cold requested) *)
	CIR_STOP_REQ	: BOOL; (* External stop request (has priority over RUN signals!) *)
	(* Physical inputs *)
	CIR_AL			: BOOL; (* Alarm input signal *)
	CIR_ST			: BOOL; (* Status input signal *)
	CIR_AUTO		: BOOL; (* Auto/Manual input signal *)
END_VAR
VAR_IN_OUT
END_VAR
VAR_OUTPUT
	(* Physical outputs *)
	CIR_EN			: BOOL;		(* CIR control output *)
	(* Status *)
	Run				: BOOL;		(* Running signal for CALs *)
	Status_Log		: BYTE;
	Status_Vis 		: DWORD;
END_VAR
VAR
	InitOK			: BOOL;
	Ctrl_Run		: BOOL;

	StartDelay		: BYTE; (* Start delay ID based to avoid peak overload *)
	StopDelay		: TOF;  (* Stop delay PLANT based for boiler heat at shutdown *)

	fCIR_AL			: FLT_TAP := ( TAP:=10, INITEV:=TRUE );
	fCIR_ST_ERR		: FLT_TAP := ( TAP:=10, INITEV:=FALSE );
	fCIR_AUTO		: FLT_TAP := ( TAP:= 5, INITEV:=TRUE );
END_VAR
(* Check initialization *)
IF NOT InitOK THEN Init(); END_IF

(* Set running flag *)
IF T_AMB<Plant_MaxRunTAmb THEN
	(* Open Control Loop [TEMPORARY] *)
	IF Ctrl_SetPoint<180 THEN Ctrl_Run:=FALSE; StartDelay:=ID;
	ELSE
		IF StartDelay>2 THEN
			Ctrl_Run:=FALSE;
			StartDelay:=StartDelay-2;
		ELSE
			Ctrl_Run:=TRUE;
		END_IF
	END_IF
	(* ==> Future obj_TERM (Thermostat) function will be an external object <== *)
ELSE
	Ctrl_Run:=FALSE;
	StartDelay:=ID;
END_IF

(* Antifreeze function: reload off delay *)
IF T_AMB<Plant_AntiFreezeTAmb THEN
	StopDelay(IN:=TRUE);
END_IF

(* Set delayed output *)
StopDelay(IN:=Ctrl_Run, PT:=Plant_CirOffDelay);
   IF CIR_STOP_REQ THEN CIR_EN:=FALSE;
ELSIF CIR_RUN_REQ  THEN CIR_EN:=TRUE;
				   ELSE CIR_EN:=StopDelay.Q; END_IF

(* Check errors *)
fCIR_AL(IN:=CIR_AL);
IF fCIR_AL.EVH THEN LogEv(EL_Alarm,EO_CAL,ID,3,'CIR_Alarm'); END_IF
IF fCIR_AL.EVL THEN LogEv(EL_Log  ,EO_CAL,ID,4,'CIR_Alarm_Recover'); END_IF

fCIR_ST_ERR(IN:=(CIR_ST<>CIR_EN));
IF fCIR_ST_ERR.EVH THEN
	IF CIR_AUTO THEN
		LogEv(SEL(CIR_ST,EL_Alarm,EL_Wrn),EO_CIR,ID,SEL(CIR_ST,5,6),'CIR_Status');
	ELSE
		LogEv(EL_Wrn,EO_CIR,ID,SEL(CIR_ST,1,2),'CIR_Manual_Wrn');
	END_IF
END_IF

fCIR_AUTO(IN:=CIR_AUTO);
IF fCIR_AUTO.EVL THEN LogEv(EL_Wrn,EO_CIR,ID,7,'CIR_Manual'); END_IF
IF fCIR_AUTO.EVH THEN LogEv(EL_Log,EO_CIR,ID,8,'CIR_Auto'  ); END_IF


(* Set RUN signal (for external objects) *)
IF fCIR_AL.OUT OR fCIR_ST_ERR.OUT THEN
	Run:=FALSE;
ELSE
	Run:=Ctrl_Run;
END_IF


(* Status color *)
   IF fCIR_AL.OUT			 				 THEN Status_Log:=2; Status_Vis:=COLOR_RED;
ELSIF fCIR_ST_ERR.OUT OR fCIR_AUTO.OUT=FALSE THEN Status_Log:=1; Status_Vis:=COLOR_YELLOW;
                  	   				 		 ELSE Status_Log:=0; Status_Vis:=SEL(CIR_EN,COLOR_GREEN_OFF,COLOR_GREEN);
END_IF
END_FUNCTION_BLOCK
ACTION Init:
(* End initialization *)
InitOK:=TRUE;
END_ACTION

(* POU Plant_Objects/obj_CRON, ST *)
FUNCTION_BLOCK obj_CRON
(* === CRONOGRAFO STANDARD ===
   v1.0[16/04/15] - Versioning
   v1.1[19/05/15] - Removed DB creation from previous year
*)
VAR_INPUT
	(* Settings *)
	ID			: BYTE;		(* Index of instanced object *)

	InitOK		: BOOL;
	Alarm		: BOOL;
	Warning		: BOOL;

	Profile		: typ_Cron_Profile; 				(* Profilo attivo *)
	ProfileNr	: BYTE;								(* Indice profilo attivo *)
	CalendarIdx : WORD;								(* Indice calendario attivo *)
	Jolly		: ARRAY[0..9] OF typ_Cron_Jolly;	(* Jolly attivi *)

END_VAR
VAR_IN_OUT
END_VAR
VAR_OUTPUT
	SetPoint		: INT;
	(* Status *)
	Status_Log		: BYTE;
	Status_Vis 		: DWORD;
END_VAR
VAR
	Buf: 	ARRAY[0..512] OF BYTE; (* AVOID THIS!! *)
	hFile: 	DWORD;
	sFile: 	STRING;
	sFile2: STRING;

	i:		WORD;
	t1:		DWORD;
	t2:		BOOL;

END_VAR
(* Check initialization *)
IF NOT InitOK THEN Init(); END_IF

(* Chrono *)
IF CalendarIdx<>Sys.Time_CT_Day THEN DB_Load(); END_IF
SetPoint:=Profile.Setpoint[Sys.Time_CT_Quarter];

(* Check jolly *)
FOR i := 0 TO 9 DO
	IF ( DT_TO_DWORD(Jolly[i].Start)>0  AND Jolly[i].End>Jolly[i].Start AND
	     Jolly[i].Start<=Sys.Time_CT_DT AND Jolly[i].End>Sys.Time_CT_DT ) THEN
			SetPoint:=Jolly[i].Temp;
	END_IF
END_FOR


(* Status color *)
   IF Alarm   THEN Status_Log:=2; Status_Vis:=COLOR_RED;
ELSIF Warning THEN Status_Log:=1; Status_Vis:=COLOR_YELLOW;
              ELSE Status_Log:=0; Status_Vis:=COLOR_GREEN;
			  END_IF
END_FUNCTION_BLOCK
ACTION DB_Create:
(*
(* Check presence of previous year *)
sFile2:=REPLACE(STR1:=sFile, STR2:=WORD_TO_STRING(Sys.Time_Year-1), L:=4, P:=LEN(FilesPath)+1);
hFile:=SysFileOpen(FileName:=sFile2, Mode:='r');
IF hFile<>0 THEN
	(* Check file version and close *)
	SysFileRead(File:=hFile, Buffer:=ADR(Buf), Size:=1);
	SysFileClose(File:=hFile);
END_IF
IF hFile<>0 AND Buf[0]=1 THEN
	(* Copy file *)
	SysFileCopy(FileDest:=sFile, FileSource:=sFile2);
ELSE
*)
	(* Create empty file *)
	hFile:=SysFileOpen(FileName:=sFile, Mode:='w');

	MEMCLR(pDestinationAddress:=ADR(Buf), BytesToClear:=SIZEOF(Buf));
	FOR i := 0 TO 10239 BY 512 DO
		t1:=SysFileWrite(File:=hFile, Buffer:=ADR(Buf), Size:=512);
	END_FOR
	Buf[0]:=1;
	t2:=SysFileSetPos(File:=hFile, Pos:=0);
	t1:=SysFileWrite(File:=hFile, Buffer:=ADR(Buf), Size:=1);
	SysFileClose(File:=hFile);
(*
END_IF
*)
END_ACTION
ACTION DB_Load:
DB_SetName();

(* Open data file *)
hFile:=SysFileOpen(FileName:=sFile, Mode:='r');

(* File not found *)
IF hFile=0 THEN
	Warning:=TRUE;
	LogEv(EL_Wrn,EO_CRON,ID,1,'No_data_file');
	DB_Create();
	(* Reopen file *)
	hFile:=SysFileOpen(FileName:=sFile, Mode:='r');
	IF hfile=0 THEN
		Alarm:=TRUE;
		LogEv(EL_Alarm,EO_CRON,ID,3,'Filesystem_error');
		RETURN;
	END_IF
END_IF

(* Check version *)
SysFileRead(File:=hFile, Buffer:=ADR(Buf), Size:=1);
IF Buf[0]<>1 THEN
	IF NOT Alarm THEN
		Alarm:=TRUE;
		LogEv(EL_Alarm,EO_CRON,ID,2,'Bad_data_version');
	END_IF
	SysFileClose(File:=hFile);
	RETURN;
END_IF

(* Read Jolly data *)
t2:=SysFileSetPos(File:=hFile, Pos:=512);
t1:=SysFileRead(File:=hFile, Buffer:=ADR(Jolly), Size:=SIZEOF(Jolly));
(* Read active profile index *)
CalendarIdx:=Sys.Time_CT_Day;
t2:=SysFileSetPos(File:=hFile, Pos:=(1024+4*CalendarIdx));
t1:=SysFileRead(File:=hFile, Buffer:=ADR(ProfileNr), Size:=SIZEOF(ProfileNr));
(* Read active profile *)
t2:=SysFileSetPos(File:=hFile, Pos:=(3072+512*ProfileNr));
t1:=SysFileRead(File:=hFile, Buffer:=ADR(Profile), Size:=SIZEOF(Profile));

(* Close file and validate data *)
SysFileClose(File:=hFile);
END_ACTION
ACTION DB_SetName:
(* Create current filename 'yyyyCRnn.DAT' *)
sFile:=CONCAT(FilesPath,WORD_TO_STRING(Sys.Time_Year));
sFile:=CONCAT(STR1:=sFile, STR2:='CR');
IF ID<10 THEN
sFile:=CONCAT(STR1:=sFile, STR2:='0');
END_IF
sFile:=CONCAT(STR1:=sFile, STR2:=BYTE_TO_STRING(ID));
sFile:=CONCAT(STR1:=sFile, STR2:='.DAT');
END_ACTION
ACTION Init:
DB_Load();
InitOK:=TRUE;
END_ACTION

(* POU Plant_Objects/obj_CRON_EDITOR, ST *)
FUNCTION_BLOCK obj_CRON_EDITOR
(* === EDITOR CRONOGRAFO ===
   v1.0[16/04/15] - Versioning
   v1.1[19/05/15] - Create empty profile when not found
*)
VAR_INPUT

	(* Common selections *)
	CN_Sel:			BYTE:=1;
	CN_Act:			BYTE;
	CN_YSel:		WORD:=2015;
	CN_YAct:		WORD;

	(* Profile editor *)
	PR_Sel: 		BYTE:=1;
	PR_Act:			BYTE;
	PR_TT:			REAL;
	PR:				typ_Cron_Profile;
	(* Profile signals *)
	PR_Load:		BOOL;
	PR_Save:		BOOL;

	(* Calendar editor *)
	CA_Sel:			BYTE:=1; (* Calendar month selected *)
	CA_Act:			BYTE;    (* Calendar month active *)
	CA_DayF:		BYTE:=0;
	CA_DayL:		BYTE:=31;
	CA_TPR:			BYTE;
	CA:				typ_Cron_Calendar; (* Only used for first 32 entries *)
	(* Calendar signals *)
	CA_Load:		BOOL;
	CA_Save:		BOOL;

	(* Jolly editor *)
	JL:				ARRAY[0..9] OF typ_Cron_Jolly;
	(* Jolly signals *)
	JL_Load:		BOOL;
	JL_Save:		BOOL;

END_VAR
VAR_OUTPUT
	Message		: STRING;
END_VAR
VAR
	sFileName	: STRING;
	sFileMode	: STRING;
	hFile		: DWORD;
	Buf			: ARRAY[0..512] OF BYTE; (* AVOID THIS!! *)

	i			: WORD;
	ver			: BYTE;
	r1			: BOOL;
	r2			: DWORD;

END_VAR
IF PR_Load THEN PR_Load_Exe(); PR_Load:=FALSE; END_IF
IF PR_Save THEN PR_Save_Exe(); PR_Save:=FALSE; END_IF
IF CA_Load THEN CA_Load_Exe(); CA_Load:=FALSE; END_IF
IF CA_Save THEN CA_Save_Exe(); CA_Save:=FALSE; END_IF
IF JL_Load THEN JL_Load_Exe(); JL_Load:=FALSE; END_IF
IF JL_Save THEN JL_Save_Exe(); JL_Save:=FALSE; END_IF
END_FUNCTION_BLOCK
ACTION CA_Load_Exe:
sFileMode:='r';
FileOpen();

IF hFile<>0 THEN

	(* Read calendar month *)
	FOR i := 0 TO 31 DO
		r1:=SysFileSetPos(File:=hFile, Pos:=(1024 + ((CA_Sel-1)*32 + i)*4));
		r2:=SysFileRead(File:=hFile, Buffer:=ADR(CA.Profile[i]), Size:=1);
	END_FOR

	(* Close file *)
	SysFileClose(File:=hFile);

	(* Validate data *)
	CA_Act :=CA_Sel;
	CN_Act :=CN_Sel;
	CN_YAct:=CN_YSel;

	Message:='Calendar load OK';

END_IF
END_ACTION
ACTION CA_Save_Exe:
sFileMode:='a';
FileOpen();

IF hFile<>0 THEN

	(* Write calendar month *)
	FOR i := 0 TO 31 DO
		r1:=SysFileSetPos(File:=hFile, Pos:=(1024 + ((CA_Sel-1)*32 + i)*4));
		r2:=SysFileGetPos(hFile);
		r2:=SysFileWrite(File:=hFile, Buffer:=ADR(CA.Profile[i]), Size:=1);
	END_FOR

	(* Close file *)
	SysFileClose(File:=hFile);

	Message:='Calendar save OK';

END_IF
END_ACTION
ACTION FileOpen:
(* Create current filename 'yyyyCRnn.DAT' *)
sFileName:=CONCAT(FilesPath,WORD_TO_STRING(CN_YSel));
sFileName:=CONCAT(STR1:=sFileName, STR2:='CR');
IF CN_Sel<10 THEN
sFileName:=CONCAT(STR1:=sFileName, STR2:='0');
END_IF
sFileName:=CONCAT(STR1:=sFileName, STR2:=BYTE_TO_STRING(CN_Sel));
sFileName:=CONCAT(STR1:=sFileName, STR2:='.DAT');

(* Check file version and size! *)
(* ... *)

(* Open data file *)
hFile:=SysFileOpen(FileName:=sFileName, Mode:='r');

(* File not found *)
IF hFile=0 THEN
	Message:='File not found - created empty file';
	(* Create empty file *)
	hFile:=SysFileOpen(FileName:=sFileName, Mode:='w');
	MEMCLR(pDestinationAddress:=ADR(Buf), BytesToClear:=SIZEOF(Buf));
	FOR i := 0 TO 10239 BY 512 DO
		SysFileWrite(File:=hFile, Buffer:=ADR(Buf), Size:=512);
	END_FOR
	Buf[0]:=1;
	SysFileSetPos(File:=hFile, Pos:=0);
	SysFileWrite(File:=hFile, Buffer:=ADR(Buf), Size:=1);
END_IF

(* Close file *)
SysFileClose(File:=hFile);

(* Open data file *)
hFile:=SysFileOpen(FileName:=sFileName, Mode:=sFileMode);
END_ACTION
ACTION JL_Load_Exe:
sFileMode:='r';
FileOpen();

IF hFile<>0 THEN

	(* Read jolly *)
	r1:=SysFileSetPos(File:=hFile, Pos:=512);
	r2:=SysFileRead(File:=hFile, Buffer:=ADR(JL), Size:=SIZEOF(JL));

	(* Close file *)
	SysFileClose(File:=hFile);

	(* Validate data *)
	CN_Act:=CN_Sel;
	CN_YAct:=CN_YSel;

	Message:='Jolly load OK';

END_IF
END_ACTION
ACTION JL_Save_Exe:
sFileMode:='a';
FileOpen();

IF hFile<>0 THEN

	(* Write selected profile *)
	r1:=SysFileSetPos(File:=hFile, Pos:=512);
	r2:=SysFileWrite(File:=hFile, Buffer:=ADR(JL), Size:=SIZEOF(JL));

	(* Close file *)
	SysFileClose(File:=hFile);

	Message:='Jolly save OK';

END_IF
END_ACTION
ACTION PR_Load_Exe:
sFileMode:='r';
FileOpen();

IF hFile<>0 THEN

	(* Read selected profile *)
	r1:=SysFileSetPos(File:=hFile, Pos:=(3072 + 512*PR_Sel));
	r2:=SysFileRead(File:=hFile, Buffer:=ADR(PR), Size:=SIZEOF(PR));

	(* Close file *)
	SysFileClose(File:=hFile);

	(* Validate data *)
	PR_Act:=PR_Sel;
	CN_Act:=CN_Sel;
	CN_YAct:=CN_YSel;

	Message:='Profile load OK';

END_IF
END_ACTION
ACTION PR_Save_Exe:
sFileMode:='a';
FileOpen();

IF hFile<>0 THEN

	(* Write selected profile *)
	r1:=SysFileSetPos(File:=hFile, Pos:=(3072 + 512*PR_Sel));
	r2:=SysFileWrite(File:=hFile, Buffer:=ADR(PR), Size:=SIZEOF(PR));

	(* Close file *)
	SysFileClose(File:=hFile);

	Message:='Profile save OK';

END_IF
END_ACTION

(* POU Plant_Objects/obj_CTL, ST *)
FUNCTION_BLOCK obj_CTL
(* === PULSE VOLUME COUNTER ===
   v1.0[16/04/15] - Versioning
*)
VAR_INPUT
	(* Settings *)
	ID				: BYTE;	(* Index of instanced object *)
	(* Physical inputs *)
	CTL_ST			: BOOL;
END_VAR
VAR_IN_OUT
	COUNT			: DWORD;
END_VAR
VAR_OUTPUT
	(* Status *)
	Status_Log		: BYTE;
END_VAR
VAR
	Filter			: FLT_TAP := ( INITEV:=FALSE );
	Timer			: TON;
	TCount			: DWORD;
	i				: DWORD;
END_VAR
(* Execute timer *)
Timer(IN:=NOT Timer.Q, PT:=T#60m);
(* Execute filter *)
Filter(IN:=CTL_ST);
(* Count event *)
IF Filter.EVH THEN
	COUNT:=COUNT+1;
	TCount:=TCount+1;
	(* Check flow rate *)
	IF TCount>=Plant_MaxWaterLoss THEN
		i:=(TCount*TIME_TO_DWORD(Timer.PT))/TIME_TO_DWORD(Timer.ET);
		LogEv(EL_AlarmStop,EO_CTL,ID,1,DWORD_TO_STRING(i));
		Status_Log:=2;
		TCount:=0;
		Timer(IN:=FALSE);
	END_IF
END_IF
(* Check timer *)
IF Timer.Q THEN
	TCount:=0;
	IF TCount<Plant_MaxWaterLoss THEN
		Status_Log:=0;
	END_IF
END_IF
END_FUNCTION_BLOCK

(* POU Plant_Objects/obj_MBUS, ST *)
FUNCTION_BLOCK obj_MBUS
(* === M-BUS PROTOCOL INTERFACE ===
   v1.0[16/03/15] - Added interface errors
*)
VAR_INPUT
	(* Settings *)
	ID				: BYTE;
	COM				: BYTE;
	BAUDRATE		: COM_BAUDRATE;
	(* Interface *)
	MBus 			: typMBus;
	MBus_Master 	: FbMBusMaster;
END_VAR
VAR_OUTPUT
	(* Status *)
	Status_Log		: BYTE;
	Status_Vis 		: DWORD;
END_VAR
VAR
	Alarm			: FLT_EVENT;
END_VAR
MBus_Master( bCOMPORT:=COM , enumBAUDRATE:=BAUDRATE , utMBus:=MBus );

(* Check status *)
Alarm(IN:=(MBus.bCOM_ERROR<>0));
IF Alarm.EVH THEN
	LogEv(EL_Alarm,EO_MBUS,ID,1,BYTE_TO_STRING(MBus.bCOM_ERROR));
END_IF
IF Alarm.EVL THEN
	LogEv(EL_Log,EO_MBUS,ID,2,'MBUS_OK');
END_IF

(* Log/visu status *)
   IF Alarm.IN   					THEN Status_Log:=2; Status_Vis:=COLOR_RED;
ELSIF (MBus.bL1_ERROR AND 16#1F)<>0 THEN Status_Log:=1; Status_Vis:=COLOR_YELLOW;
  				 					ELSE Status_Log:=0; Status_Vis:=COLOR_GREEN;
END_IF
END_FUNCTION_BLOCK

(* POU Plant_Objects/obj_MBUS_CTB, ST *)
FUNCTION_BLOCK obj_MBUS_CTB
(* === MBUS HEAT CONTABILIZER ===
   v1.0[16/04/15] - Versioning
*)
VAR_INPUT
	(* Settings *)
	ID				: BYTE;
	ADDRESS			: BYTE;
	(* Controls *)
	UpdateNow		: BOOL;
END_VAR
VAR_IN_OUT
	MBus			: typMBus;
END_VAR
VAR_OUTPUT
	(* Visu/Log *)
	Status_Log		: BYTE;
	Status_Vis 		: DWORD;
END_VAR
VAR
	T1			: TON := ( PT:=T#120s );
	M1			: FbMBus_Heat;
	M1_Start	: BOOL;
	C1			: FbUnitConverter;
END_VAR
(* Auto refresh timer *)
T1( IN:=NOT ( T1.Q OR M1_Start ) );
(* Trigger refresh *)
IF NOT M1_Start AND (T1.Q OR UpdateNow) THEN
	M1_Start:=TRUE;
	UpdateNow:=FALSE;
END_IF

M1(
	dwAdr:=ADDRESS,
	xSND_NKE:=TRUE ,
	utMBus:=MBus ,
	xStart:=M1_Start ,
);


(* Check status *)
IF M1.bError<>0 THEN Status_Log:=2; Status_Vis:=COLOR_RED;
			    ELSE Status_Log:=0; Status_Vis:=COLOR_GREEN;
END_IF
END_FUNCTION_BLOCK

(* POU Plant_Objects/obj_MODBUS, ST *)
FUNCTION_BLOCK obj_MODBUS
(* === MODBUS PROTOCOL INTERFACE ===
   v1.0[16/03/15] - Support for RS485 half-duplex
				  - Rewritten vars management with state machine
   v1.1[27/03/15] - Fixed vars manager & introduced retry before alarm
   v1.2[16/04/15] - Changed initialization alarm to a simple warning
   v1.3[20/04/15] - Var alarm auto-recover when succesful reading of last error variable
*)
VAR CONSTANT
	VARS_Max	: BYTE := 32;
END_VAR
VAR_INPUT
	(* Settings *)
	ID			: BYTE;
	COM			: BYTE;
	BAUDRATE	: COM_BAUDRATE;
	RS485		: BOOL := FALSE;
	(* Interface *)
	MB_MASTER	: MODBUS_EXTENDED_MASTER;
	MB_Start	: BOOL;
	MB_Query	: typModbusExtendedQuery;
	MB_Resp		: typModbusResponse;
	MB_Lock		: BOOL;
	(* Variables management *)
	VARS_En		: BOOL;
	VARS		: ARRAY [0..VARS_Max] OF typ_MODBUS_VAR;
	VARS_Check	: BOOL;
	VARS_Alarm	: BOOL;
END_VAR
VAR_OUTPUT
	(* Status *)
	Status_Log	: BYTE;
	Status_Vis	: DWORD;
END_VAR
VAR
	i			: BYTE;
	Alarm		: FLT_EVENT;
	VarTmr		: TON := (PT:=T#1s);
	VarSta		: BYTE; (* Status *)
	VarCnt		: BYTE; (* Scan counter *)
	VarRetry	: BYTE;
	VarAlarm	: BYTE; (* Last variable with errors *)
END_VAR
MB_MASTER(
	ENABLE:=TRUE ,
	ASCII_Mode:=FALSE,
	bCOM_PORT:=COM ,
	cbCOM_BAUDRATE:=BAUDRATE ,
	cpCOM_PARITY:=PARITY_NO ,
	csCOM_STOPBITS:=STOPBITS_1 ,
	cbsCOM_BYTESIZE:=BS_8 ,
	cfCOM_FLOW_CONTROL:=SEL(RS485,NO_FLOW_CONTROL,HALFDUPLEX) ,
	tTIME_OUT:=t#250ms ,
	StartFunction:=MB_Start ,
	ExtQuery:=MB_Query ,
	Response:=MB_Resp  );

(* Process variable management *)
IF VARS_En THEN VARS_Process(); END_IF

(* Check status *)
Alarm(IN:=(MB_MASTER.bInterfaceError<>0));
IF Alarm.EVH THEN
	LogEv(SEL(MB_MASTER.bInterfaceError<>3,EL_Wrn,EL_Alarm),EO_MODBUS,ID,1,BYTE_TO_STRING(MB_MASTER.bInterfaceError));
END_IF
IF Alarm.EVL THEN
	LogEv(EL_Log,EO_MODBUS,ID,2,'MODBUS_OK');
END_IF

(* Log/visu status *)
   IF Alarm.IN   THEN Status_Log:=2; Status_Vis:=COLOR_RED;
ELSIF Vars_Alarm THEN Status_Log:=1; Status_Vis:=COLOR_YELLOW;
  				 ELSE Status_Log:=0; Status_Vis:=COLOR_GREEN;
END_IF
END_FUNCTION_BLOCK
ACTION VARS_Process:
(* Update var timers *)
VarTmr(IN:=(NOT VarTmr.Q));
IF VarTmr.Q THEN
	FOR i := 0 TO VARS_Max DO
		IF VARS[i].Refresh_Cnt>0 THEN VARS[i].Refresh_Cnt:=VARS[i].Refresh_Cnt-1; END_IF
	END_FOR
	VARS_Check:=TRUE;
END_IF


(* Process status *)
CASE VarSta OF
	0: (* === Init *)
		VarCnt:=0;
		VarSta:=1;

	1: (* === Wait check signal *)
		IF VARS_Check THEN
			VARS_Check:=FALSE;
			VarCnt:=0;
			VarSta:=2;
		END_IF

	2: (* === Check loop *)
		IF NOT (MB_Lock OR MB_Start) THEN
			WHILE VarCnt<=VARS_Max AND VarSta=2 DO
				(* Check only active vars *)
				IF VARS[VarCnt].SlaveAddress<>0 THEN
					(* Check var auto-refresh on timer checks *)
					IF VARS[VarCnt].Refresh_Time>0 AND VARS[VarCnt].Refresh_Cnt=0 THEN
						VARS[VarCnt].Refresh_Cnt:=VARS[VarCnt].Refresh_Time;
						VarSta:=3;
					END_IF
					(* Check refresh for change or request *)
					CASE VARS[VarCnt].FunCode OF
						16#5,16#6,16#F,16#10:
							IF VARS[VarCnt].Variable^<>VARS[VarCnt].Variable_Mirror THEN
								VARS[VarCnt].Variable_Mirror:=VARS[VarCnt].Variable^;
								VarSta:=3;
							END_IF
						16#1,16#2,16#3,16#4:
							IF VARS[VarCnt].Variable_Mirror<>0 THEN
								VARS[VarCnt].Variable_Mirror:=0;
								VarSta:=3;
							END_IF
					END_CASE
				END_IF
				(* Process query *)
				IF VarSta=3 THEN
					MB_Lock:=TRUE;
					MB_Query.SlaveAddress:=VARS[VarCnt].SlaveAddress;
					MB_Query.FunctionCode:=VARS[VarCnt].FunCode;
					CASE VARS[VarCnt].FunCode OF
						16#5,16#6,16#F,16#10:
							MB_Query.Read_StartAddress:=0;
							MB_Query.Read_Quantity:=0;
							MB_Query.Write_StartAddress:=VARS[VarCnt].FunAddress;
							MB_Query.Write_Quantity:=VARS[VarCnt].Variable_Size;
							MB_Query.Write_Data[0]:=VARS[VarCnt].Variable^;
						16#1,16#2,16#3,16#4:
							MB_Query.Read_StartAddress:=VARS[VarCnt].FunAddress;
							IF VARS[VarCnt].Variable_Size=200 THEN MB_Query.Read_Quantity:=2; ELSE
							  MB_Query.Read_Quantity:=VARS[VarCnt].Variable_Size;
							END_IF
							MB_Query.Write_StartAddress:=0;
							MB_Query.Write_Quantity:=0;
					END_CASE
					VarRetry:=0;
					MB_Start:=TRUE;
				ELSE
					VarCnt:=VarCnt+1;
				END_IF
			END_WHILE
			(* Check loop completed -> no actions *)
			IF VarSta=2 THEN VarSta:=1; END_IF
		END_IF

	3: (* === Wait & process MB response *)
		IF NOT MB_Start THEN
			IF MB_MASTER.MB_Error=0 THEN
				CASE VARS[VarCnt].FunCode OF
					16#1,16#2,16#3,16#4:
						IF VARS[VarCnt].Variable_Size=200 THEN
							COPY_32SWAP16(ADR(MB_Resp.Data), VARS[VarCnt].Variable);
						ELSIF VARS[VarCnt].Variable_Size>1 THEN
							MEMCPY(ADR(MB_Resp.Data), VARS[VarCnt].Variable, 2*VARS[VarCnt].Variable_Size);
						ELSE
							VARS[VarCnt].Variable^:=MB_Resp.Data[0];
						END_IF
				END_CASE
				MB_Lock:=FALSE;
				(* Signal error recovery *)
				IF VARS_Alarm=TRUE AND VarCnt=VarAlarm THEN
					LogEv(EL_Wrn,EO_MODBUS,ID,5,'');
					VARS_Alarm:=FALSE;
				END_IF
				(* Next var *)
				VarCnt:=VarCnt+1;
				VarSta:=2;
			ELSE
				IF VarRetry<3 THEN
					VarRetry:=VarRetry+1;
					MB_Start:=TRUE;
				ELSE
					MB_Lock:=FALSE;
					(* Signal error *)
					IF VARS_Alarm=FALSE THEN
						LogEv(EL_Wrn,EO_MODBUS,ID,3,INT_TO_STRING(MB_MASTER.MB_Error));
						VARS_Alarm:=TRUE;
						VarAlarm:=VarCnt-1;
					END_IF
					(* Next var *)
					VarCnt:=VarCnt+1;
					VarSta:=2;
				END_IF
			END_IF
		END_IF

ELSE
	VarSta:=0;
END_CASE
END_ACTION

(* POU Plant_Objects/obj_MODBUS_ROBUR_DDC, ST *)
FUNCTION_BLOCK obj_MODBUS_ROBUR_DDC
(* === MODBUS ROBUR DDC MAIN CONTROLLER ===
   v1.0[16/04/15] - Versioning
*)
VAR_INPUT
	(* Settings *)
	ID				: BYTE;
	NetID			: WORD; (* Network ID on ROBUR DDC *)

	(* Controls *)
	Run				: BOOL;

	(* MODBUS data to CAL *)
	En				: WORD; (* 00006 *)
	SetPoint		: WORD;	(* 40577 *)
	Log_ReadAck		: WORD; (* 40202 , Write GRU01_Log_Count *)
	Reset_UnitID	: WORD; (* 40244 *)
	Reset_Request	: WORD; (* 40245 *)

	(* MODBUS data from CAL *)
	TSend			: INT; 	(* 30253 *)
	TRet			: INT; 	(* 30254 *)
	TAmb			: INT;	(* 30255 *)
	ActSetPoint		: INT;  (* 30680 *)
	Status			: WORD; (* 30965 { 0:OK, 1=INF, 2=WRN, 3=ERR } *)

	Log_Count		: WORD; (* 40001 *)
	Log_Sta			: BYTE;					(* Current status of processed error record *)
	Log_Record		: ARRAY [0..4] OF WORD; (* 40011 + Idx*5 *)
	Log_Record_Rq	: BOOL;
	Reset_Status	: WORD; (* 40246 *)

END_VAR
VAR_IN_OUT
	Clima 			: typ_Clima;
	MODBUS			: obj_MODBUS;
END_VAR
VAR_OUTPUT
	(* Visu/Log *)
	Status_Log		: BYTE;
	Status_Vis : DWORD;
END_VAR
VAR
	InitOK		: BOOL;
	Alarm		: BOOL;
	AlarmBUS	: BOOL;
	Warning		: BOOL;

	Curve 		: CHARCURVE;
	Curve_Err 	: BYTE;
	Curve_Temp	: INT;

	s1 : STRING;
	i  : WORD;
	ec : BOOL;

END_VAR
(* Check initialization *)
IF NOT InitOK THEN Init(); END_IF

(* Check MODBUS connection *)
IF MODBUS.VARS_Alarm THEN
	IF NOT AlarmBUS THEN
		LogEv(EL_Alarm,EO_GRU,ID,5,'');
		AlarmBUS:=TRUE;
	END_IF
ELSE
	AlarmBUS:=FALSE;
END_IF

(* Check LOGS *)
Log_Check();

(* Check DDC state *)
IF Status=3 THEN
	IF NOT Alarm THEN
		Alarm:=TRUE;
		LogEv(EL_Alarm,EO_GRU,ID,6,'');
	END_IF
ELSE
	Alarm:=FALSE;
END_IF

(* Check climatic setup *)
IF NOT Clima.InitOK THEN Clima_Default(); END_IF;
(* Calculate Setpoint *)
Curve(	IN:= T_AMB,	N:= 5, P:= Clima.Points,
		OUT=> Curve_Temp, ERR=> Curve_Err );
IF Curve_Err>0 THEN
	IF NOT Warning THEN
		Warning:=TRUE;
		LogEv(EL_Wrn,EO_GRU,ID,2,'GRU_Climatic_Error');
	END_IF
ELSE
	Warning:=FALSE;
END_IF

(* Send temperature set-point (force update every 1min) *)
SetPoint:=Curve_Temp;

(* Attivazione caldaia *)
IF Run THEN
	En:=1;
ELSE
	En:=0;
END_IF

(* Check rearm flags *)
Reset_Check();

(* Status color *)
   IF Alarm OR AlarmBUS  	  THEN Status_Log:=2; Status_Vis:=COLOR_RED;
ELSIF Warning OR Status=2     THEN Status_Log:=1; Status_Vis:=COLOR_YELLOW;
              				  ELSE Status_Log:=0; Status_Vis:=SEL(Run,COLOR_GREEN_OFF,COLOR_GREEN);
END_IF
END_FUNCTION_BLOCK
ACTION Clima_Default:
Clima.Points[0].X:=-300; Clima.Points[0].Y:=650;
Clima.Points[1].X:=-50 ; Clima.Points[1].Y:=650;
Clima.Points[2].X:= 200; Clima.Points[2].Y:=200;
Clima.Points[3].X:= 300; Clima.Points[3].Y:=200;
Clima.Points[4].X:= 500; Clima.Points[4].Y:=200;
Clima.InitOK:=TRUE;
LogEv(EL_Wrn,EO_GRU,ID,1,'GRU_Climatic_default');
END_ACTION
ACTION Init:
(* 00002 - Write master enable *)
MODBUS.VARS[0].SlaveAddress:=1;
MODBUS.VARS[0].FunCode:=16#F;
MODBUS.VARS[0].FunAddress:=16#1;
MODBUS.VARS[0].Refresh_Time:=120;
MODBUS.VARS[0].Variable:=ADR(En);
MODBUS.VARS[0].Variable_Size:=1;
MODBUS.VARS[0].Variable_Mirror:=0;
(* 40577 -  Write master Setpoint *)
MODBUS.VARS[1].SlaveAddress:=1;
MODBUS.VARS[1].FunCode:=16#6;
MODBUS.VARS[1].FunAddress:=16#240;
MODBUS.VARS[1].Refresh_Time:=120;
MODBUS.VARS[1].Variable:=ADR(SetPoint);
MODBUS.VARS[1].Variable_Size:=1;
MODBUS.VARS[1].Variable_Mirror:=0;
(* 40202 - Write acknowledge for errors *)
MODBUS.VARS[2].SlaveAddress:=1;
MODBUS.VARS[2].FunCode:=16#6;
MODBUS.VARS[2].FunAddress:=16#C9;
MODBUS.VARS[2].Refresh_Time:=0;
MODBUS.VARS[2].Variable:=ADR(Log_ReadAck);
MODBUS.VARS[2].Variable_Size:=1;
MODBUS.VARS[2].Variable_Mirror:=0;

(* 30253 - Read master TSend *)
MODBUS.VARS[3].SlaveAddress:=1;
MODBUS.VARS[3].FunCode:=16#4;
MODBUS.VARS[3].FunAddress:=16#FC;
MODBUS.VARS[3].Refresh_Time:=10;
MODBUS.VARS[3].Variable:=ADR(TSend);
MODBUS.VARS[3].Variable_Size:=1;
MODBUS.VARS[3].Variable_Mirror:=1; (* <== Refresh at startup *)
(* 30254 - Read master TRet *)
MODBUS.VARS[4].SlaveAddress:=1;
MODBUS.VARS[4].FunCode:=16#4;
MODBUS.VARS[4].FunAddress:=16#FD;
MODBUS.VARS[4].Refresh_Time:=10;
MODBUS.VARS[4].Variable:=ADR(TRet);
MODBUS.VARS[4].Variable_Size:=1;
MODBUS.VARS[4].Variable_Mirror:=1; (* <== Refresh at startup *)
(* 30255 - Read master TAmbient *)
MODBUS.VARS[5].SlaveAddress:=1;
MODBUS.VARS[5].FunCode:=16#4;
MODBUS.VARS[5].FunAddress:=16#FE;
MODBUS.VARS[5].Refresh_Time:=10;
MODBUS.VARS[5].Variable:=ADR(TAmb);
MODBUS.VARS[5].Variable_Size:=1;
MODBUS.VARS[5].Variable_Mirror:=1; (* <== Refresh at startup *)
(* 30680 - Read master active SetPoint *)
MODBUS.VARS[6].SlaveAddress:=1;
MODBUS.VARS[6].FunCode:=16#4;
MODBUS.VARS[6].FunAddress:=16#02A7;
MODBUS.VARS[6].Refresh_Time:=10;
MODBUS.VARS[6].Variable:=ADR(ActSetPoint);
MODBUS.VARS[6].Variable_Size:=1;
MODBUS.VARS[6].Variable_Mirror:=0;
(* 30965 - Read master general alarm *)
MODBUS.VARS[7].SlaveAddress:=1;
MODBUS.VARS[7].FunCode:=16#4;
MODBUS.VARS[7].FunAddress:=16#03C4;
MODBUS.VARS[7].Refresh_Time:=10;
MODBUS.VARS[7].Variable:=ADR(Status);
MODBUS.VARS[7].Variable_Size:=1;
MODBUS.VARS[7].Variable_Mirror:=0;

(* 40001 - Read pending logs *)
MODBUS.VARS[8].SlaveAddress:=1;
MODBUS.VARS[8].FunCode:=16#3;
MODBUS.VARS[8].FunAddress:=16#0;
MODBUS.VARS[8].Refresh_Time:=10;
MODBUS.VARS[8].Variable:=ADR(Log_Count);
MODBUS.VARS[8].Variable_Size:=1;
MODBUS.VARS[8].Variable_Mirror:=0;
(* 40011 - Read 1st log entry *)
MODBUS.VARS[9].SlaveAddress:=1;
MODBUS.VARS[9].FunCode:=16#3;
MODBUS.VARS[9].FunAddress:=16#A;
MODBUS.VARS[9].Refresh_Time:=0;
MODBUS.VARS[9].Variable:=ADR(Log_Record);
MODBUS.VARS[9].Variable_Size:=5;
MODBUS.VARS[9].Variable_Mirror:=0;

(****************************************** PDC01 *******)
(* 12028 + 64*ID *)
MODBUS.VARS[10].SlaveAddress:=1;
MODBUS.VARS[10].FunCode:=16#2;
MODBUS.VARS[10].FunAddress:=16#07EB + 64*0;
MODBUS.VARS[10].Refresh_Time:=20;
MODBUS.VARS[10].Variable:=ADR(PDC01.OnOff);
MODBUS.VARS[10].Variable_Size:=1;
MODBUS.VARS[10].Variable_Mirror:=0;
(* 35023 + 250*ID *)
MODBUS.VARS[11].SlaveAddress:=1;
MODBUS.VARS[11].FunCode:=16#4;
MODBUS.VARS[11].FunAddress:=16#139E + 250*0;
MODBUS.VARS[11].Refresh_Time:=20;
MODBUS.VARS[11].Variable:=ADR(PDC01.TSend);
MODBUS.VARS[11].Variable_Size:=1;
MODBUS.VARS[11].Variable_Mirror:=0;
(* 35024 + 250*ID *)
MODBUS.VARS[12].SlaveAddress:=1;
MODBUS.VARS[12].FunCode:=16#4;
MODBUS.VARS[12].FunAddress:=16#139F + 250*0;
MODBUS.VARS[12].Refresh_Time:=20;
MODBUS.VARS[12].Variable:=ADR(PDC01.TRet);
MODBUS.VARS[12].Variable_Size:=1;
MODBUS.VARS[12].Variable_Mirror:=0;
(* 35041 + 250*ID *)
MODBUS.VARS[13].SlaveAddress:=1;
MODBUS.VARS[13].FunCode:=16#4;
MODBUS.VARS[13].FunAddress:=16#13B0 + 250*0;
MODBUS.VARS[13].Refresh_Time:=20;
MODBUS.VARS[13].Variable:=ADR(PDC01.Flow);
MODBUS.VARS[13].Variable_Size:=1;
MODBUS.VARS[13].Variable_Mirror:=0;
(* 35044 + 250*ID *)
MODBUS.VARS[14].SlaveAddress:=1;
MODBUS.VARS[14].FunCode:=16#4;
MODBUS.VARS[14].FunAddress:=16#13B3 + 250*0;
MODBUS.VARS[14].Refresh_Time:=20;
MODBUS.VARS[14].Variable:=ADR(PDC01.Power);
MODBUS.VARS[14].Variable_Size:=1;
MODBUS.VARS[14].Variable_Mirror:=0;
(* 35061 + 250*ID *)
MODBUS.VARS[15].SlaveAddress:=1;
MODBUS.VARS[15].FunCode:=16#4;
MODBUS.VARS[15].FunAddress:=16#13C4 + 250*0;
MODBUS.VARS[15].Refresh_Time:=20;
MODBUS.VARS[15].Variable:=ADR(PDC01.Status);
MODBUS.VARS[15].Variable_Size:=1;
MODBUS.VARS[15].Variable_Mirror:=0;

(****************************************** CAL01 *******)
(* 12028 + 64*ID *)
MODBUS.VARS[16].SlaveAddress:=1;
MODBUS.VARS[16].FunCode:=16#2;
MODBUS.VARS[16].FunAddress:=16#07EB + 64*1;
MODBUS.VARS[16].Refresh_Time:=20;
MODBUS.VARS[16].Variable:=ADR(CAL01.OnOff);
MODBUS.VARS[16].Variable_Size:=1;
MODBUS.VARS[16].Variable_Mirror:=0;
(* 35023 + 250*ID *)
MODBUS.VARS[17].SlaveAddress:=1;
MODBUS.VARS[17].FunCode:=16#4;
MODBUS.VARS[17].FunAddress:=16#139E + 250*1;
MODBUS.VARS[17].Refresh_Time:=20;
MODBUS.VARS[17].Variable:=ADR(CAL01.TSend);
MODBUS.VARS[17].Variable_Size:=1;
MODBUS.VARS[17].Variable_Mirror:=0;
(* 35024 + 250*ID *)
MODBUS.VARS[18].SlaveAddress:=1;
MODBUS.VARS[18].FunCode:=16#4;
MODBUS.VARS[18].FunAddress:=16#139F + 250*1;
MODBUS.VARS[18].Refresh_Time:=20;
MODBUS.VARS[18].Variable:=ADR(CAL01.TRet);
MODBUS.VARS[18].Variable_Size:=1;
MODBUS.VARS[18].Variable_Mirror:=0;
(* 35061 + 250*ID *)
MODBUS.VARS[19].SlaveAddress:=1;
MODBUS.VARS[19].FunCode:=16#4;
MODBUS.VARS[19].FunAddress:=16#13C4 + 250*1;
MODBUS.VARS[19].Refresh_Time:=20;
MODBUS.VARS[19].Variable:=ADR(CAL01.Status);
MODBUS.VARS[19].Variable_Size:=1;
MODBUS.VARS[19].Variable_Mirror:=0;

(****************************************** CAL02*******)
(* 12028 + 64*ID *)
MODBUS.VARS[20].SlaveAddress:=1;
MODBUS.VARS[20].FunCode:=16#2;
MODBUS.VARS[20].FunAddress:=16#07EB + 64*2;
MODBUS.VARS[20].Refresh_Time:=20;
MODBUS.VARS[20].Variable:=ADR(CAL02.OnOff);
MODBUS.VARS[20].Variable_Size:=1;
MODBUS.VARS[20].Variable_Mirror:=0;
(* 35023 + 250*ID *)
MODBUS.VARS[21].SlaveAddress:=1;
MODBUS.VARS[21].FunCode:=16#4;
MODBUS.VARS[21].FunAddress:=16#139E + 250*2;
MODBUS.VARS[21].Refresh_Time:=20;
MODBUS.VARS[21].Variable:=ADR(CAL02.TSend);
MODBUS.VARS[21].Variable_Size:=1;
MODBUS.VARS[21].Variable_Mirror:=0;
(* 35024 + 250*ID *)
MODBUS.VARS[22].SlaveAddress:=1;
MODBUS.VARS[22].FunCode:=16#4;
MODBUS.VARS[22].FunAddress:=16#139F + 250*2;
MODBUS.VARS[22].Refresh_Time:=20;
MODBUS.VARS[22].Variable:=ADR(CAL02.TRet);
MODBUS.VARS[22].Variable_Size:=1;
MODBUS.VARS[22].Variable_Mirror:=0;
(* 35061 + 250*ID *)
MODBUS.VARS[23].SlaveAddress:=1;
MODBUS.VARS[23].FunCode:=16#4;
MODBUS.VARS[23].FunAddress:=16#13C4 + 250*2;
MODBUS.VARS[23].Refresh_Time:=20;
MODBUS.VARS[23].Variable:=ADR(CAL02.Status);
MODBUS.VARS[23].Variable_Size:=1;
MODBUS.VARS[23].Variable_Mirror:=0;

(****************************************** REARM*******)
(* 40244(W) - Reset UnitID *)
MODBUS.VARS[24].SlaveAddress:=1;
MODBUS.VARS[24].FunCode:=16#6;
MODBUS.VARS[24].FunAddress:=16#F3;
MODBUS.VARS[24].Refresh_Time:=0;
MODBUS.VARS[24].Variable:=ADR(Reset_UnitID);
MODBUS.VARS[24].Variable_Size:=1;
MODBUS.VARS[24].Variable_Mirror:=0;
(* 40245(W) - Reset Request *)
MODBUS.VARS[25].SlaveAddress:=1;
MODBUS.VARS[25].FunCode:=16#6;
MODBUS.VARS[25].FunAddress:=16#F4;
MODBUS.VARS[25].Refresh_Time:=0;
MODBUS.VARS[25].Variable:=ADR(Reset_Request);
MODBUS.VARS[25].Variable_Size:=1;
MODBUS.VARS[25].Variable_Mirror:=0;
(* 40246(R) - Status of Reset *)
MODBUS.VARS[26].SlaveAddress:=1;
MODBUS.VARS[26].FunCode:=16#3;
MODBUS.VARS[26].FunAddress:=16#F5;
MODBUS.VARS[26].Refresh_Time:=0;
MODBUS.VARS[26].Variable:=ADR(Reset_Status);
MODBUS.VARS[26].Variable_Size:=1;
MODBUS.VARS[26].Variable_Mirror:=0;


(* Enable variables control *)
MODBUS.VARS_En:=TRUE;
(* End initialization *)
InitOK:=TRUE;
END_ACTION
ACTION Log_Check:
IF Log_Count>0 THEN
	IF Log_Sta=0 THEN
		(* Request log record *)
		MODBUS.VARS[9].Variable_Mirror:=1;
		Log_Sta:=1;
	ELSIF Log_Sta=1 THEN
		(* Check log reading *)
		IF MODBUS.VARS[9].Variable_Mirror=0 AND MODBUS.VarSta=1 THEN
			(* Generate LogEv *)
			Log_Send();
			(* Ack reading *)
			Log_ReadAck:=1;
			MODBUS.VARS[2].Variable_Mirror:=0;
			Log_Sta:=2;
		END_IF
	ELSIF Log_Sta=2 THEN
		(* Check ack writing *)
		IF MODBUS.VARS[2].Variable_Mirror=1 AND MODBUS.VarSta=1 THEN
			(* Update log count *)
			MODBUS.VARS[8].Variable_Mirror:=1;
			Log_Sta:=3;
		END_IF
	ELSIF Log_Sta=3 THEN
		(* Check ack reading *)
		IF MODBUS.VARS[8].Variable_Mirror=0 AND MODBUS.VarSta=1 THEN
			Log_Sta:=0;
		END_IF
	END_IF
ELSE
	Log_Sta:=0;
END_IF
END_ACTION
ACTION Log_Send:
(* Generate debug log *)
s1:=RAWTOHEXSTR(pData:=ADR(Log_Record), DataLen:=SIZEOF(Log_Record));
LogEv(EL_Log,EO_GRU,ID,10,s1);

